C03634=1069.661,411.759,-112.459,175.801,35.006,156.496
C03635=1069.668,412.006,-112.501,175.806,35.015,156.498
C03636=1069.676,412.252,-112.545,175.812,35.025,156.501
C03637=1069.684,412.498,-112.589,175.818,35.034,156.503
C03638=1069.691,412.744,-112.631,175.824,35.044,156.505
C03639=1069.699,412.990,-112.675,175.831,35.054,156.508
C03640=1069.707,413.237,-112.719,175.837,35.064,156.510
C03641=1069.715,413.514,-112.768,175.844,35.074,156.512
C03642=1069.725,413.793,-112.817,175.850,35.085,156.515
C03643=1069.734,414.072,-112.867,175.857,35.096,156.518
C03644=1069.742,414.350,-112.916,175.864,35.108,156.520
C03645=1069.751,414.596,-112.959,175.870,35.117,156.523
C03646=1069.759,414.842,-113.003,175.877,35.127,156.525
C03647=1069.766,415.088,-113.047,175.883,35.137,156.527
C03648=1069.774,415.334,-113.091,175.888,35.147,156.530
C03649=1069.782,415.580,-113.135,175.894,35.157,156.532
C03650=1069.789,415.826,-113.178,175.901,35.167,156.535
C03651=1069.797,416.072,-113.222,175.907,35.177,156.537
C03652=1069.804,416.319,-113.267,175.913,35.187,156.539
C03653=1069.813,416.564,-113.311,175.919,35.197,156.542
C03654=1069.820,416.811,-113.354,175.926,35.208,156.544
C03655=1069.828,417.056,-113.399,175.932,35.218,156.547
C03656=1069.836,417.302,-113.443,175.938,35.228,156.549
C03657=1069.844,417.549,-113.487,175.944,35.238,156.552
C03658=1069.852,417.794,-113.531,175.951,35.248,156.554
C03659=1069.860,418.040,-113.575,175.957,35.259,156.557
C03660=1069.868,418.286,-113.620,175.963,35.269,156.559
C03661=1069.875,418.532,-113.664,175.970,35.279,156.562
C03662=1069.883,418.778,-113.708,175.976,35.290,156.564
C03663=1069.892,419.024,-113.753,175.983,35.300,156.567
C03664=1069.900,419.270,-113.797,175.989,35.310,156.569
C03665=1069.908,419.515,-113.841,175.995,35.321,156.572
C03666=1069.916,419.761,-113.886,176.003,35.331,156.574
C03667=1069.924,420.007,-113.930,176.009,35.342,156.577
C03668=1069.932,420.254,-113.975,176.016,35.353,156.579
C03669=1069.940,420.499,-114.020,176.022,35.363,156.582
C03670=1069.948,420.745,-114.064,176.029,35.373,156.584
C03671=1069.956,420.991,-114.108,176.035,35.384,156.587
C03672=1069.964,421.238,-114.154,176.042,35.395,156.590
C03673=1069.972,421.483,-114.199,176.048,35.406,156.592
C03674=1069.980,421.729,-114.243,176.055,35.417,156.595
C03675=1069.988,421.975,-114.288,176.062,35.427,156.598
C03676=1069.996,422.220,-114.333,176.069,35.438,156.600
C03677=1070.004,422.466,-114.378,176.075,35.449,156.603
C03678=1070.012,422.712,-114.423,176.082,35.460,156.606
C03679=1070.020,422.957,-114.468,176.088,35.471,156.608
C03680=1070.028,423.203,-114.513,176.095,35.482,156.611
C03681=1070.037,423.449,-114.558,176.102,35.493,156.614
C03682=1070.044,423.695,-114.604,176.109,35.504,156.616
C03683=1070.052,423.940,-114.648,176.115,35.515,156.619
C03684=1070.061,424.187,-114.694,176.122,35.526,156.622
C03685=1070.069,424.432,-114.739,176.130,35.537,156.625
C03686=1070.076,424.678,-114.784,176.136,35.548,156.627
C03687=1070.085,424.924,-114.829,176.143,35.559,156.630
C03688=1070.093,425.169,-114.875,176.150,35.571,156.633
C03689=1070.102,425.415,-114.920,176.157,35.582,156.636
C03690=1070.110,425.660,-114.966,176.164,35.593,156.638
C03691=1070.118,425.907,-115.011,176.171,35.604,156.641
C03692=1070.126,426.152,-115.056,176.177,35.615,156.644
C03693=1070.135,426.398,-115.102,176.185,35.627,156.647
C03694=1070.143,426.643,-115.148,176.192,35.638,156.650
C03695=1070.152,426.889,-115.193,176.199,35.650,156.652
C03696=1070.159,427.135,-115.239,176.206,35.661,156.655
C03697=1070.170,427.431,-115.294,176.214,35.675,156.659
C03698=1070.179,427.729,-115.350,176.223,35.689,156.662
C03699=1070.190,428.026,-115.405,176.232,35.703,156.666
C03700=1070.199,428.324,-115.461,176.240,35.717,156.669
C03701=1070.208,428.570,-115.507,176.248,35.729,156.672
C03702=1070.217,428.815,-115.553,176.255,35.741,156.675
C03703=1070.224,429.061,-115.599,176.263,35.753,156.678
C03704=1070.233,429.306,-115.645,176.270,35.764,156.681
C03705=1070.241,429.552,-115.691,176.277,35.776,156.684
C03706=1070.250,429.797,-115.737,176.285,35.788,156.687
C03707=1070.258,430.043,-115.783,176.291,35.800,156.690
C03708=1070.267,430.288,-115.830,176.299,35.812,156.693
C03709=1070.275,430.534,-115.877,176.306,35.824,156.696
C03710=1070.283,430.779,-115.922,176.314,35.836,156.699
C03711=1070.292,431.025,-115.968,176.321,35.848,156.702
C03712=1070.301,431.270,-116.015,176.329,35.860,156.705
C03713=1070.309,431.516,-116.061,176.336,35.872,156.708
C03714=1070.318,431.762,-116.108,176.344,35.884,156.711
C03715=1070.326,432.007,-116.155,176.352,35.896,156.714
C03716=1070.334,432.252,-116.201,176.359,35.909,156.717
C03717=1070.343,432.498,-116.248,176.367,35.922,156.721
C03718=1070.351,432.743,-116.294,176.374,35.934,156.724
C03719=1070.360,432.989,-116.341,176.382,35.946,156.727
C03720=1070.368,433.234,-116.388,176.390,35.959,156.730
C03721=1070.377,433.479,-116.435,176.397,35.971,156.733
C03722=1070.386,433.725,-116.482,176.406,35.984,156.736
C03723=1070.393,433.970,-116.529,176.414,35.996,156.739
C03724=1070.402,434.216,-116.576,176.421,36.009,156.743
C03725=1070.411,434.461,-116.623,176.429,36.021,156.746
C03726=1070.419,434.706,-116.670,176.437,36.034,156.749
C03727=1070.428,434.952,-116.717,176.444,36.047,156.752
C03728=1070.437,435.197,-116.764,176.452,36.059,156.756
C03729=1070.445,435.442,-116.811,176.461,36.072,156.759
C03730=1070.454,435.687,-116.859,176.468,36.085,156.762
C03731=1070.463,435.933,-116.905,176.476,36.098,156.765
C03732=1070.471,436.178,-116.953,176.484,36.111,156.769
C03733=1070.480,436.423,-117.001,176.493,36.124,156.772
C03734=1070.489,436.669,-117.048,176.501,36.137,156.775
C03735=1070.498,436.914,-117.095,176.508,36.150,156.779
C03736=1070.506,437.159,-117.143,176.516,36.163,156.782
C03737=1070.515,437.404,-117.190,176.525,36.176,156.785
C03738=1070.525,437.649,-117.238,176.533,36.189,156.789
C03739=1070.533,437.894,-117.286,176.541,36.202,156.792
C03740=1070.541,438.140,-117.333,176.550,36.215,156.796
C03741=1070.551,438.386,-117.381,176.558,36.229,156.799
C03742=1070.560,438.630,-117.428,176.566,36.242,156.802
C03743=1070.568,438.875,-117.477,176.574,36.255,156.806
C03744=1070.578,439.121,-117.525,176.582,36.269,156.809
C03745=1070.586,439.365,-117.572,176.591,36.282,156.813
C03746=1070.595,439.611,-117.620,176.599,36.295,156.816
C03747=1070.604,439.856,-117.668,176.608,36.309,156.820
C03748=1070.612,440.101,-117.717,176.616,36.323,156.823
C03749=1070.622,440.346,-117.764,176.625,36.336,156.827
C03750=1070.631,440.591,-117.812,176.633,36.350,156.830
C03751=1070.640,440.837,-117.861,176.642,36.364,156.834
C03752=1070.649,441.082,-117.908,176.650,36.377,156.838
C03753=1070.657,441.314,-117.955,176.659,36.391,156.841
C03754=1070.665,441.548,-118.001,176.667,36.404,156.845
C03755=1070.674,441.781,-118.047,176.675,36.417,156.848
C03756=1070.683,442.015,-118.093,176.683,36.430,156.851
C03757=1070.692,442.248,-118.140,176.693,36.444,156.855
C03758=1070.700,442.481,-118.186,176.701,36.457,156.858
C03759=1070.708,442.715,-118.232,176.709,36.471,156.862
C03760=1070.717,442.948,-118.279,176.718,36.484,156.865
C03761=1070.727,443.193,-118.327,176.726,36.498,156.869
C03762=1070.736,443.438,-118.376,176.735,36.513,156.873
C03763=1070.745,443.682,-118.425,176.744,36.527,156.877
C03764=1070.754,443.927,-118.474,176.754,36.541,156.881
C03765=1070.764,444.172,-118.522,176.762,36.556,156.884
C03766=1070.773,444.418,-118.571,176.771,36.570,156.888
C03767=1070.781,444.662,-118.620,176.781,36.584,156.892
C03768=1070.790,444.908,-118.669,176.790,36.599,156.896
C03769=1070.800,445.152,-118.719,176.799,36.614,156.900
C03770=1070.809,445.397,-118.768,176.808,36.628,156.904
C03771=1070.819,445.642,-118.817,176.817,36.643,156.907
C03772=1070.828,445.887,-118.867,176.826,36.658,156.911
C03773=1070.837,446.132,-118.915,176.836,36.672,156.915
C03774=1070.846,446.376,-118.965,176.845,36.687,156.919
C03775=1070.855,446.621,-119.014,176.855,36.702,156.923
C03776=1070.864,446.866,-119.064,176.864,36.717,156.927
C03777=1070.874,447.111,-119.113,176.874,36.732,156.931
C03778=1070.884,447.355,-119.163,176.883,36.747,156.935
C03779=1070.893,447.601,-119.212,176.893,36.762,156.939
C03780=1070.903,447.846,-119.262,176.902,36.777,156.943
C03781=1070.913,448.089,-119.312,176.911,36.793,156.947
C03782=1070.922,448.332,-119.360,176.920,36.807,156.951
C03783=1070.932,448.577,-119.410,176.929,36.822,156.955
C03784=1070.944,448.821,-119.458,176.937,36.836,156.959
C03785=1070.957,449.066,-119.505,176.945,36.850,156.963
C03786=1070.972,449.311,-119.551,176.953,36.863,156.966
C03787=1070.987,449.556,-119.598,176.960,36.876,156.970
C03788=1071.004,449.802,-119.643,176.968,36.888,156.973
C03789=1070.654,449.802,-119.894,176.954,37.029,157.010
C03790=1070.638,449.556,-119.849,176.947,37.016,157.007
C03791=1070.622,449.311,-119.803,176.939,37.004,157.004
C03792=1070.608,449.066,-119.756,176.931,36.990,157.000
C03793=1070.595,448.821,-119.709,176.923,36.977,156.996
C03794=1070.582,448.576,-119.661,176.914,36.963,156.993
C03795=1070.571,448.332,-119.612,176.905,36.948,156.989
C03796=1070.562,448.088,-119.563,176.896,36.933,156.985
C03797=1070.553,447.845,-119.513,176.886,36.918,156.981
C03798=1070.543,447.601,-119.463,176.877,36.903,156.977
C03799=1070.533,447.356,-119.413,176.867,36.888,156.973
C03800=1070.523,447.111,-119.364,176.858,36.873,156.969
C03801=1070.514,446.866,-119.315,176.848,36.858,156.965
C03802=1070.505,446.621,-119.265,176.838,36.843,156.961
C03803=1070.496,446.376,-119.215,176.829,36.828,156.957
C03804=1070.486,446.131,-119.166,176.819,36.814,156.953
C03805=1070.477,445.887,-119.116,176.810,36.799,156.949
C03806=1070.468,445.641,-119.067,176.800,36.784,156.945
C03807=1070.458,445.397,-119.018,176.792,36.770,156.941
C03808=1070.449,445.153,-118.969,176.782,36.755,156.937
C03809=1070.440,444.908,-118.920,176.773,36.741,156.933
C03810=1070.431,444.663,-118.870,176.764,36.726,156.929
C03811=1070.422,444.417,-118.821,176.754,36.711,156.925
C03812=1070.412,444.173,-118.772,176.745,36.697,156.922
C03813=1070.403,443.928,-118.723,176.736,36.683,156.918
C03814=1070.394,443.683,-118.674,176.727,36.668,156.914
C03815=1070.384,443.438,-118.626,176.718,36.654,156.910
C03816=1070.375,443.193,-118.577,176.708,36.640,156.906
C03817=1070.366,442.949,-118.528,176.700,36.626,156.903
C03818=1070.358,442.724,-118.484,176.692,36.612,156.899
C03819=1070.349,442.500,-118.439,176.684,36.600,156.896
C03820=1070.341,442.276,-118.394,176.675,36.587,156.892
C03821=1070.333,442.052,-118.351,176.667,36.574,156.889
C03822=1070.324,441.828,-118.306,176.659,36.562,156.886
C03823=1070.316,441.604,-118.261,176.651,36.549,156.882
C03824=1070.308,441.380,-118.218,176.643,36.536,156.879
C03825=1070.300,441.156,-118.173,176.635,36.524,156.876
C03826=1070.291,440.912,-118.124,176.627,36.510,156.872
C03827=1070.282,440.666,-118.076,176.618,36.496,156.869
C03828=1070.273,440.421,-118.027,176.609,36.482,156.865
C03829=1070.264,440.176,-117.980,176.600,36.468,156.861
C03830=1070.254,439.931,-117.931,176.592,36.455,156.858
C03831=1070.246,439.686,-117.883,176.583,36.442,156.854
C03832=1070.237,439.441,-117.836,176.575,36.428,156.851
C03833=1070.228,439.195,-117.787,176.566,36.415,156.847
C03834=1070.219,438.951,-117.739,176.558,36.401,156.844
C03835=1070.210,438.705,-117.692,176.549,36.388,156.840
C03836=1070.202,438.460,-117.643,176.541,36.374,156.837
C03837=1070.193,438.215,-117.596,176.533,36.361,156.833
C03838=1070.183,437.969,-117.548,176.524,36.348,156.830
C03839=1070.174,437.724,-117.501,176.516,36.335,156.827
C03840=1070.166,437.480,-117.453,176.507,36.322,156.823
C03841=1070.157,437.234,-117.405,176.499,36.309,156.820
C03842=1070.148,436.989,-117.357,176.491,36.296,156.817
C03843=1070.139,436.744,-117.310,176.483,36.283,156.813
C03844=1070.130,436.498,-117.263,176.475,36.270,156.810
C03845=1070.121,436.253,-117.215,176.467,36.257,156.807
C03846=1070.112,436.008,-117.168,176.459,36.244,156.803
C03847=1070.104,435.762,-117.121,176.450,36.231,156.800
C03848=1070.096,435.517,-117.073,176.442,36.218,156.797
C03849=1070.087,435.272,-117.026,176.434,36.205,156.793
C03850=1070.078,435.027,-116.979,176.427,36.193,156.790
C03851=1070.069,434.781,-116.931,176.419,36.180,156.787
C03852=1070.060,434.536,-116.885,176.410,36.167,156.784
C03853=1070.051,434.291,-116.837,176.402,36.155,156.780
C03854=1070.043,434.045,-116.790,176.395,36.142,156.777
C03855=1070.034,433.800,-116.744,176.387,36.130,156.774
C03856=1070.026,433.554,-116.697,176.379,36.117,156.771
C03857=1070.017,433.309,-116.649,176.371,36.105,156.768
C03858=1070.008,433.064,-116.603,176.364,36.092,156.764
C03859=1070.001,432.818,-116.555,176.356,36.080,156.761
C03860=1069.992,432.572,-116.509,176.348,36.068,156.758
C03861=1069.984,432.328,-116.462,176.341,36.055,156.755
C03862=1069.976,432.082,-116.416,176.333,36.043,156.752
C03863=1069.967,431.837,-116.369,176.325,36.031,156.749
C03864=1069.958,431.591,-116.322,176.318,36.018,156.746
C03865=1069.950,431.346,-116.275,176.310,36.006,156.743
C03866=1069.941,431.100,-116.229,176.303,35.994,156.740
C03867=1069.932,430.855,-116.183,176.295,35.982,156.737
C03868=1069.924,430.609,-116.137,176.287,35.970,156.734
C03869=1069.916,430.364,-116.090,176.280,35.958,156.730
C03870=1069.907,430.118,-116.043,176.272,35.946,156.727
C03871=1069.898,429.873,-115.998,176.265,35.934,156.724
C03872=1069.890,429.627,-115.951,176.257,35.923,156.721
C03873=1069.882,429.382,-115.905,176.250,35.910,156.718
C03874=1069.874,429.136,-115.859,176.242,35.899,156.716
C03875=1069.865,428.891,-115.812,176.235,35.887,156.713
C03876=1069.857,428.645,-115.767,176.228,35.875,156.710
C03877=1069.849,428.399,-115.721,176.221,35.864,156.707
C03878=1069.838,428.100,-115.665,176.212,35.849,156.703
C03879=1069.829,427.801,-115.609,176.203,35.835,156.700
C03880=1069.818,427.503,-115.553,176.194,35.821,156.696
C03881=1069.808,427.203,-115.497,176.185,35.807,156.693
C03882=1069.800,426.957,-115.451,176.178,35.796,156.690
C03883=1069.791,426.712,-115.406,176.171,35.784,156.687
C03884=1069.783,426.466,-115.360,176.164,35.773,156.684
C03885=1069.775,426.220,-115.315,176.156,35.761,156.681
C03886=1069.766,425.974,-115.269,176.150,35.750,156.678
C03887=1069.758,425.729,-115.224,176.142,35.739,156.676
C03888=1069.750,425.483,-115.178,176.135,35.728,156.673
C03889=1069.741,425.238,-115.133,176.129,35.716,156.670
C03890=1069.733,424.992,-115.087,176.121,35.705,156.667
C03891=1069.725,424.747,-115.042,176.114,35.694,156.665
C03892=1069.717,424.501,-114.996,176.108,35.683,156.662
C03893=1069.709,424.255,-114.951,176.101,35.672,156.659
C03894=1069.701,424.009,-114.906,176.093,35.661,156.656
C03895=1069.692,423.764,-114.860,176.087,35.650,156.654
C03896=1069.685,423.517,-114.815,176.080,35.639,156.651
C03897=1069.676,423.272,-114.770,176.073,35.628,156.648
C03898=1069.667,423.027,-114.725,176.066,35.617,156.645
C03899=1069.660,422.780,-114.680,176.060,35.606,156.643
C03900=1069.652,422.535,-114.635,176.053,35.595,156.640
C03901=1069.644,422.289,-114.590,176.045,35.584,156.637
C03902=1069.635,422.043,-114.545,176.039,35.573,156.635
C03903=1069.628,421.797,-114.500,176.032,35.563,156.632
C03904=1069.620,421.552,-114.455,176.026,35.552,156.629
C03905=1069.611,421.306,-114.410,176.019,35.541,156.627
C03906=1069.604,421.060,-114.365,176.012,35.530,156.624
C03907=1069.595,420.814,-114.321,176.005,35.520,156.622
C03908=1069.587,420.568,-114.276,175.999,35.509,156.619
C03909=1069.579,420.322,-114.232,175.993,35.499,156.616
C03910=1069.571,420.076,-114.187,175.986,35.488,156.614
C03911=1069.563,419.831,-114.142,175.980,35.477,156.611
C03912=1069.555,419.585,-114.097,175.973,35.467,156.609
C03913=1069.547,419.339,-114.053,175.966,35.457,156.606
C03914=1069.539,419.093,-114.009,175.959,35.446,156.604
C03915=1069.530,418.846,-113.965,175.953,35.436,156.601
C03916=1069.522,418.601,-113.920,175.947,35.426,156.599
C03917=1069.515,418.355,-113.875,175.940,35.416,156.596
C03918=1069.507,418.109,-113.831,175.934,35.405,156.594
C03919=1069.499,417.863,-113.787,175.928,35.395,156.591
C03920=1069.491,417.617,-113.742,175.921,35.384,156.589
C03921=1069.483,417.371,-113.699,175.915,35.374,156.586
C03922=1069.475,417.125,-113.654,175.909,35.364,156.584
C03923=1069.467,416.879,-113.610,175.902,35.354,156.581
C03924=1069.459,416.633,-113.566,175.896,35.344,156.579
C03925=1069.451,416.387,-113.522,175.890,35.334,156.576
C03926=1069.444,416.141,-113.477,175.883,35.323,156.574
C03927=1069.437,415.896,-113.434,175.876,35.313,156.571
C03928=1069.429,415.650,-113.390,175.870,35.304,156.569
C03929=1069.421,415.404,-113.346,175.864,35.293,156.567
C03930=1069.413,415.158,-113.302,175.859,35.284,156.564
C03931=1069.405,414.911,-113.258,175.851,35.274,156.562
C03932=1069.397,414.665,-113.214,175.846,35.264,156.560
C03933=1069.389,414.419,-113.170,175.840,35.254,156.557
C03934=1069.380,414.139,-113.121,175.832,35.243,156.554
C03935=1069.371,413.859,-113.071,175.825,35.232,156.552
C03936=1069.362,413.579,-113.021,175.818,35.220,156.549
C03937=1069.353,413.298,-112.972,175.811,35.210,156.546
C03938=1069.346,413.053,-112.928,175.805,35.200,156.544
C03939=1069.337,412.807,-112.885,175.799,35.190,156.542
C03940=1069.329,412.561,-112.842,175.793,35.180,156.540
C03941=1069.322,412.314,-112.798,175.788,35.171,156.537
C03942=1069.314,412.069,-112.755,175.782,35.162,156.535
C03943=1069.306,411.823,-112.712,175.776,35.152,156.533
C03944=1069.298,411.576,-112.668,175.770,35.142,156.530
C03945=1069.290,411.330,-112.625,175.764,35.133,156.528
C03946=1069.284,411.084,-112.582,175.757,35.123,156.526
C03947=1069.275,410.838,-112.539,175.751,35.113,156.524
C03948=1069.267,410.591,-112.495,175.745,35.104,156.521
C03949=1069.260,410.346,-112.452,175.740,35.095,156.519
C03950=1069.252,410.099,-112.409,175.734,35.085,156.517
C03951=1069.245,409.853,-112.367,175.728,35.076,156.515
C03952=1069.237,409.607,-112.323,175.722,35.067,156.513
C03953=1069.230,409.361,-112.280,175.716,35.057,156.510
C03954=1069.222,409.115,-112.237,175.710,35.048,156.508
C03955=1069.214,408.868,-112.194,175.704,35.039,156.506
C03956=1069.207,408.622,-112.151,175.699,35.030,156.504
C03957=1069.199,408.376,-112.108,175.693,35.020,156.502
C03958=1069.191,408.130,-112.065,175.687,35.011,156.499
C03959=1069.184,407.884,-112.023,175.682,35.002,156.497
C03960=1069.176,407.637,-111.980,175.676,34.993,156.495
C03961=1069.169,407.392,-111.937,175.671,34.984,156.493
C03962=1069.161,407.145,-111.895,175.665,34.975,156.491
C03963=1069.154,406.899,-111.851,175.659,34.966,156.489
C03964=1069.146,406.652,-111.808,175.653,34.956,156.486
C03965=1069.139,406.406,-111.766,175.648,34.948,156.484
C03966=1069.132,406.161,-111.723,175.642,34.938,156.482
C03967=1069.123,405.914,-111.681,175.636,34.930,156.480
C03968=1069.117,405.668,-111.638,175.631,34.921,156.478
C03969=1069.109,405.422,-111.596,175.626,34.912,156.476
C03970=1069.102,405.175,-111.554,175.620,34.903,156.474
C03971=1069.094,404.929,-111.512,175.614,34.894,156.472
C03972=1069.086,404.683,-111.470,175.608,34.885,156.470
C03973=1069.079,404.436,-111.427,175.603,34.876,156.468
C03974=1069.071,404.190,-111.385,175.598,34.868,156.466
C03975=1069.064,403.943,-111.342,175.592,34.859,156.464
C03976=1069.056,403.697,-111.300,175.587,34.850,156.462
C03977=1069.049,403.451,-111.258,175.581,34.841,156.460
C03978=1069.042,403.204,-111.215,175.575,34.833,156.458
C03979=1069.034,402.959,-111.173,175.570,34.824,156.455
C03980=1069.027,402.713,-111.132,175.565,34.815,156.453
C03981=1069.018,402.466,-111.089,175.559,34.807,156.451
C03982=1069.012,402.219,-111.047,175.553,34.798,156.449
C03983=1069.004,401.973,-111.005,175.549,34.790,156.447
C03984=1068.997,401.727,-110.964,175.543,34.781,156.445
C03985=1068.989,401.481,-110.922,175.537,34.773,156.444
C03986=1068.981,401.234,-110.880,175.532,34.764,156.442
C03987=1068.974,400.987,-110.837,175.527,34.756,156.440
C03988=1068.967,400.741,-110.796,175.521,34.747,156.438
C03989=1068.959,400.495,-110.754,175.516,34.739,156.436
C03990=1068.951,400.219,-110.707,175.510,34.729,156.434
C03991=1068.943,399.942,-110.661,175.504,34.719,156.431
C03992=1068.935,399.666,-110.614,175.498,34.710,156.429
C03993=1068.926,399.390,-110.567,175.492,34.701,156.427
C03994=1068.919,399.143,-110.526,175.487,34.693,156.425
C03995=1068.912,398.897,-110.484,175.482,34.684,156.423
C03996=1068.904,398.651,-110.442,175.476,34.676,156.421
C03997=1068.897,398.404,-110.401,175.472,34.668,156.419
C03998=1068.889,398.158,-110.359,175.466,34.660,156.417
C03999=1068.882,397.912,-110.318,175.460,34.651,156.416
C04000=1068.875,397.665,-110.277,175.456,34.643,156.414
C04001=1068.867,397.418,-110.235,175.450,34.635,156.412
C04002=1068.860,397.172,-110.194,175.445,34.627,156.410
C04003=1068.853,396.926,-110.152,175.440,34.618,156.408
C04004=1068.846,396.680,-110.111,175.434,34.611,156.406
C04005=1068.839,396.433,-110.070,175.430,34.602,156.404
C04006=1068.831,396.187,-110.029,175.424,34.594,156.402
C04007=1068.824,395.940,-109.988,175.420,34.586,156.401
C04008=1068.817,395.694,-109.947,175.414,34.578,156.399
C04009=1068.809,395.447,-109.905,175.409,34.570,156.397
C04010=1068.801,395.201,-109.865,175.404,34.562,156.395
C04011=1068.795,394.955,-109.824,175.399,34.554,156.393
C04012=1068.787,394.708,-109.783,175.394,34.546,156.391
C04013=1068.780,394.462,-109.741,175.389,34.538,156.390
C04014=1068.773,394.215,-109.700,175.384,34.531,156.388
C04015=1068.766,393.969,-109.659,175.378,34.522,156.386
C04016=1068.759,393.722,-109.619,175.374,34.515,156.384
C04017=1068.751,393.476,-109.578,175.368,34.507,156.383
C04018=1068.744,393.229,-109.537,175.364,34.499,156.381
C04019=1068.737,392.983,-109.496,175.358,34.491,156.379
C04020=1068.730,392.736,-109.455,175.353,34.484,156.377
C04021=1068.722,392.490,-109.415,175.348,34.476,156.376
C04022=1068.716,392.244,-109.374,175.343,34.468,156.374
C04023=1068.709,391.997,-109.333,175.338,34.460,156.372
C04024=1068.701,391.750,-109.293,175.334,34.453,156.370
C04025=1068.694,391.504,-109.252,175.328,34.445,156.369
C04026=1068.687,391.257,-109.211,175.324,34.437,156.367
C04027=1068.679,391.011,-109.171,175.318,34.429,156.365
C04028=1068.672,390.764,-109.131,175.314,34.422,156.363
C04029=1068.665,390.518,-109.089,175.309,34.414,156.362
C04030=1068.658,390.272,-109.050,175.304,34.407,156.360
C04031=1068.651,390.025,-109.009,175.299,34.399,156.358
C04032=1068.643,389.778,-108.969,175.294,34.392,156.356
C04033=1068.637,389.532,-108.929,175.289,34.384,156.355
C04034=1068.629,389.285,-108.888,175.284,34.376,156.353
C04035=1068.622,389.039,-108.848,175.279,34.369,156.351
C04036=1068.615,388.792,-108.808,175.274,34.361,156.350
C04037=1068.607,388.546,-108.768,175.270,34.354,156.348
C04038=1068.600,388.299,-108.727,175.264,34.346,156.346
C04039=1068.592,388.052,-108.687,175.260,34.339,156.345
C04040=1068.586,387.806,-108.647,175.255,34.332,156.343
C04041=1068.579,387.559,-108.608,175.250,34.325,156.341
C04042=1068.571,387.313,-108.568,175.246,34.317,156.340
C04043=1068.564,387.067,-108.527,175.240,34.310,156.338
C04044=1068.557,386.820,-108.487,175.236,34.302,156.337
C04045=1068.550,386.573,-108.447,175.231,34.295,156.335
C04046=1068.542,386.313,-108.405,175.226,34.287,156.333
C04047=1068.535,386.052,-108.363,175.221,34.279,156.331
C04048=1068.528,385.792,-108.320,175.216,34.272,156.330
C04049=1068.521,385.532,-108.278,175.211,34.264,156.328
C04050=1068.513,385.285,-108.239,175.206,34.257,156.326
C04051=1068.506,385.038,-108.199,175.201,34.250,156.325
C04052=1068.499,384.792,-108.159,175.197,34.243,156.323
C04053=1068.492,384.546,-108.119,175.192,34.235,156.322
C04054=1068.485,384.301,-108.079,175.188,34.228,156.320
C04055=1068.478,384.056,-108.041,175.182,34.221,156.318
C04056=1068.471,383.811,-108.001,175.178,34.214,156.317
C04057=1068.464,383.567,-107.962,175.174,34.207,156.315
C04058=1068.458,383.322,-107.922,175.168,34.200,156.314
C04059=1068.450,383.078,-107.883,175.164,34.193,156.312
C04060=1068.444,382.833,-107.844,175.160,34.186,156.311
C04061=1068.436,382.588,-107.804,175.155,34.179,156.309
C04062=1068.430,382.342,-107.764,175.151,34.171,156.307
C04063=1068.423,382.095,-107.725,175.146,34.165,156.306
C04064=1068.416,381.849,-107.686,175.141,34.157,156.304
C04065=1068.409,381.601,-107.646,175.137,34.151,156.303
C04066=1068.402,381.355,-107.607,175.132,34.143,156.301
C04067=1068.396,381.108,-107.568,175.127,34.137,156.300
C04068=1068.388,380.862,-107.528,175.123,34.129,156.298
C04069=1068.381,380.614,-107.489,175.118,34.123,156.297
C04070=1068.374,380.368,-107.449,175.114,34.116,156.295
C04071=1068.367,380.121,-107.411,175.109,34.109,156.294
C04072=1068.360,379.874,-107.372,175.104,34.102,156.292
C04073=1068.353,379.628,-107.332,175.100,34.095,156.291
C04074=1068.346,379.381,-107.293,175.096,34.088,156.289
C04075=1068.339,379.134,-107.254,175.090,34.081,156.288
C04076=1068.332,378.888,-107.215,175.086,34.075,156.286
C04077=1068.325,378.641,-107.176,175.082,34.068,156.285
C04078=1068.318,378.394,-107.137,175.077,34.061,156.283
C04079=1068.311,378.147,-107.098,175.073,34.054,156.282
C04080=1068.305,377.900,-107.059,175.068,34.048,156.280
C04081=1068.297,377.654,-107.020,175.064,34.041,156.279
C04082=1068.290,377.407,-106.980,175.059,34.034,156.277
C04083=1068.283,377.160,-106.942,175.055,34.027,156.276
C04084=1068.276,376.913,-106.903,175.051,34.021,156.274
C04085=1068.270,376.666,-106.864,175.046,34.014,156.273
C04086=1068.263,376.419,-106.825,175.041,34.007,156.271
C04087=1068.256,376.172,-106.786,175.037,34.001,156.270
C04088=1068.249,375.926,-106.747,175.032,33.994,156.268
C04089=1068.242,375.679,-106.709,175.028,33.987,156.267
C04090=1068.236,375.432,-106.670,175.024,33.981,156.266
C04091=1068.229,375.185,-106.631,175.020,33.974,156.264
C04092=1068.222,374.938,-106.592,175.015,33.967,156.263
C04093=1068.215,374.691,-106.554,175.011,33.961,156.261
C04094=1068.209,374.444,-106.515,175.007,33.954,156.260
C04095=1068.202,374.197,-106.476,175.001,33.947,156.258
C04096=1068.195,373.951,-106.438,174.997,33.941,156.257
C04097=1068.188,373.705,-106.400,174.993,33.934,156.256
C04098=1068.182,373.464,-106.362,174.989,33.928,156.254
C04099=1068.175,373.223,-106.324,174.984,33.922,156.253
C04100=1068.169,372.983,-106.286,174.980,33.915,156.251
C04101=1068.162,372.742,-106.250,174.976,33.909,156.250
C04102=1068.155,372.501,-106.212,174.972,33.903,156.249
C04103=1068.148,372.261,-106.175,174.967,33.896,156.247
C04104=1068.141,372.020,-106.138,174.963,33.890,156.246
C04105=1068.135,371.780,-106.100,174.959,33.884,156.245
C04106=1068.128,371.533,-106.062,174.955,33.878,156.243
C04107=1068.121,371.286,-106.024,174.950,33.871,156.242
C04108=1068.114,371.039,-105.986,174.946,33.865,156.241
C04109=1068.107,370.792,-105.947,174.942,33.859,156.239
C04110=1068.101,370.545,-105.909,174.938,33.853,156.238
C04111=1068.093,370.298,-105.871,174.933,33.846,156.237
C04112=1068.087,370.051,-105.833,174.929,33.840,156.235
C04113=1068.080,369.805,-105.795,174.925,33.833,156.234
C04114=1068.073,369.558,-105.757,174.921,33.827,156.232
C04115=1068.067,369.310,-105.719,174.917,33.821,156.231
C04116=1068.059,369.064,-105.680,174.912,33.814,156.230
C04117=1068.053,368.816,-105.642,174.908,33.808,156.228
C04118=1068.046,368.570,-105.605,174.904,33.802,156.227
C04119=1068.040,368.322,-105.567,174.900,33.796,156.226
C04120=1068.033,368.076,-105.528,174.895,33.790,156.224
C04121=1068.026,367.828,-105.491,174.891,33.784,156.223
C04122=1068.020,367.582,-105.453,174.887,33.777,156.222
C04123=1068.012,367.335,-105.415,174.883,33.771,156.220
C04124=1068.006,367.087,-105.377,174.879,33.765,156.219
C04125=1067.999,366.841,-105.340,174.874,33.758,156.218
C04126=1067.992,366.594,-105.301,174.870,33.753,156.217
C04127=1067.985,366.347,-105.264,174.866,33.746,156.215
C04128=1067.979,366.100,-105.226,174.862,33.740,156.214
C04129=1067.972,365.853,-105.188,174.857,33.734,156.213
C04130=1067.966,365.605,-105.150,174.853,33.728,156.211
C04131=1067.959,365.359,-105.113,174.849,33.722,156.210
C04132=1067.952,365.112,-105.075,174.845,33.715,156.209
C04133=1067.946,364.865,-105.038,174.841,33.710,156.207
C04134=1067.939,364.618,-105.000,174.838,33.703,156.206
C04135=1067.932,364.370,-104.963,174.833,33.698,156.205
C04136=1067.926,364.123,-104.925,174.829,33.691,156.204
C04137=1067.919,363.876,-104.888,174.825,33.686,156.202
C04138=1067.912,363.629,-104.850,174.821,33.679,156.201
C04139=1067.906,363.382,-104.812,174.817,33.674,156.200
C04140=1067.899,363.135,-104.775,174.812,33.667,156.198
C04141=1067.892,362.888,-104.738,174.808,33.662,156.197
C04142=1067.885,362.641,-104.701,174.804,33.656,156.196
C04143=1067.879,362.394,-104.663,174.800,33.649,156.195
C04144=1067.872,362.146,-104.626,174.796,33.644,156.193
C04145=1067.865,361.899,-104.589,174.793,33.638,156.192
C04146=1067.858,361.653,-104.552,174.788,33.632,156.191
C04147=1067.852,361.405,-104.514,174.784,33.626,156.190
C04148=1067.846,361.158,-104.477,174.780,33.620,156.188
C04149=1067.839,360.910,-104.440,174.776,33.614,156.187
C04150=1067.832,360.664,-104.403,174.772,33.609,156.186
C04151=1067.825,360.417,-104.366,174.768,33.603,156.185
C04152=1067.819,360.170,-104.329,174.763,33.596,156.184
C04153=1067.812,359.922,-104.291,174.760,33.591,156.182
C04154=1067.805,359.692,-104.257,174.756,33.586,156.181
C04155=1067.800,359.463,-104.223,174.752,33.580,156.180
C04156=1067.794,359.233,-104.189,174.749,33.575,156.179
C04157=1067.788,359.003,-104.154,174.745,33.569,156.178
C04158=1067.782,358.773,-104.119,174.742,33.564,156.177
C04159=1067.776,358.543,-104.085,174.737,33.558,156.176
C04160=1067.769,358.313,-104.051,174.733,33.553,156.174
C04161=1067.763,358.084,-104.016,174.730,33.548,156.173
C04162=1067.757,357.837,-103.979,174.726,33.542,156.172
C04163=1067.750,357.589,-103.943,174.722,33.536,156.171
C04164=1067.743,357.342,-103.906,174.718,33.531,156.170
C04165=1067.736,357.095,-103.869,174.715,33.525,156.169
C04166=1067.730,356.848,-103.832,174.710,33.519,156.167
C04167=1067.723,356.600,-103.796,174.706,33.514,156.166
C04168=1067.717,356.353,-103.759,174.702,33.508,156.165
C04169=1067.710,356.106,-103.723,174.698,33.502,156.164
C04170=1067.703,355.858,-103.686,174.695,33.497,156.163
C04171=1067.697,355.611,-103.649,174.691,33.491,156.162
C04172=1067.690,355.364,-103.612,174.687,33.485,156.160
C04173=1067.684,355.117,-103.576,174.683,33.480,156.159
C04174=1067.677,354.870,-103.539,174.678,33.474,156.158
C04175=1067.671,354.623,-103.502,174.675,33.469,156.157
C04176=1067.664,354.375,-103.466,174.671,33.463,156.156
C04177=1067.657,354.128,-103.430,174.667,33.457,156.154
C04178=1067.650,353.881,-103.393,174.663,33.452,156.153
C04179=1067.644,353.634,-103.357,174.660,33.446,156.152
C04180=1067.638,353.387,-103.320,174.656,33.440,156.151
C04181=1067.631,353.139,-103.284,174.652,33.435,156.150
C04182=1067.624,352.892,-103.247,174.647,33.429,156.149
C04183=1067.618,352.644,-103.211,174.644,33.424,156.148
C04184=1067.612,352.397,-103.175,174.640,33.418,156.146
C04185=1067.605,352.150,-103.138,174.636,33.413,156.145
C04186=1067.599,351.903,-103.102,174.633,33.407,156.144
C04187=1067.592,351.656,-103.066,174.629,33.402,156.143
C04188=1067.586,351.408,-103.030,174.625,33.397,156.142
C04189=1067.579,351.161,-102.994,174.621,33.391,156.141
C04190=1067.572,350.913,-102.957,174.618,33.386,156.140
C04191=1067.565,350.667,-102.921,174.613,33.380,156.138
C04192=1067.559,350.419,-102.885,174.609,33.374,156.137
C04193=1067.553,350.172,-102.849,174.605,33.369,156.136
C04194=1067.546,349.924,-102.814,174.602,33.364,156.135
C04195=1067.539,349.677,-102.777,174.598,33.358,156.134
C04196=1067.533,349.430,-102.740,174.594,33.353,156.133
C04197=1067.526,349.182,-102.705,174.591,33.348,156.132
C04198=1067.520,348.935,-102.669,174.587,33.342,156.131
C04199=1067.514,348.688,-102.633,174.583,33.337,156.130
C04200=1067.507,348.440,-102.597,174.580,33.331,156.129
C04201=1067.501,348.193,-102.562,174.576,33.326,156.127
C04202=1067.494,347.946,-102.525,174.571,33.321,156.126
C04203=1067.488,347.698,-102.489,174.568,33.316,156.125
C04204=1067.481,347.451,-102.453,174.564,33.310,156.124
C04205=1067.475,347.203,-102.417,174.560,33.304,156.123
C04206=1067.467,346.957,-102.382,174.557,33.299,156.122
C04207=1067.461,346.709,-102.346,174.553,33.294,156.121
C04208=1067.455,346.461,-102.310,174.549,33.289,156.120
C04209=1067.448,346.214,-102.274,174.546,33.283,156.119
C04210=1067.442,345.986,-102.242,174.542,33.279,156.118
C04211=1067.436,345.758,-102.209,174.539,33.273,156.117
C04212=1067.431,345.531,-102.176,174.536,33.269,156.116
C04213=1067.425,345.303,-102.143,174.532,33.264,156.115
C04214=1067.419,345.074,-102.110,174.529,33.259,156.114
C04215=1067.413,344.846,-102.078,174.525,33.254,156.113
C04216=1067.407,344.619,-102.044,174.521,33.249,156.112
C04217=1067.401,344.390,-102.012,174.518,33.245,156.111
C04218=1067.395,344.143,-101.976,174.514,33.239,156.110
C04219=1067.388,343.895,-101.941,174.511,33.234,156.109
C04220=1067.382,343.648,-101.905,174.507,33.229,156.108
C04221=1067.375,343.400,-101.870,174.504,33.224,156.107
C04222=1067.368,343.154,-101.834,174.500,33.218,156.105
C04223=1067.363,342.907,-101.799,174.496,33.213,156.104
C04224=1067.356,342.659,-101.764,174.493,33.208,156.103
C04225=1067.349,342.412,-101.728,174.489,33.203,156.102
C04226=1067.343,342.164,-101.693,174.486,33.198,156.101
C04227=1067.336,341.917,-101.658,174.482,33.192,156.100
C04228=1067.330,341.670,-101.622,174.478,33.188,156.099
C04229=1067.324,341.422,-101.587,174.475,33.182,156.098
C04230=1067.317,341.175,-101.552,174.471,33.177,156.097
C04231=1067.310,340.927,-101.517,174.468,33.172,156.096
C04232=1067.304,340.679,-101.481,174.464,33.167,156.095
C04233=1067.298,340.431,-101.446,174.460,33.162,156.094
C04234=1067.291,340.184,-101.411,174.456,33.157,156.093
C04235=1067.285,339.937,-101.376,174.452,33.152,156.092
C04236=1067.279,339.690,-101.341,174.449,33.146,156.091
C04237=1067.272,339.442,-101.306,174.445,33.142,156.090
C04238=1067.265,339.194,-101.271,174.442,33.136,156.089
C04239=1067.259,338.947,-101.235,174.438,33.132,156.088
C04240=1067.253,338.699,-101.200,174.435,33.126,156.087
C04241=1067.246,338.453,-101.166,174.431,33.121,156.086
C04242=1067.241,338.204,-101.130,174.428,33.116,156.085
C04243=1067.234,337.957,-101.095,174.424,33.111,156.084
C04244=1067.227,337.710,-101.060,174.421,33.106,156.083
C04245=1067.221,337.462,-101.026,174.417,33.101,156.082
C04246=1067.215,337.215,-100.991,174.414,33.096,156.081
C04247=1067.208,336.967,-100.955,174.410,33.091,156.080
C04248=1067.202,336.719,-100.921,174.407,33.086,156.079
C04249=1067.195,336.472,-100.886,174.403,33.081,156.078
C04250=1067.189,336.225,-100.852,174.400,33.076,156.077
C04251=1067.183,335.977,-100.817,174.396,33.071,156.076
C04252=1067.176,335.729,-100.782,174.393,33.066,156.075
C04253=1067.169,335.482,-100.747,174.389,33.061,156.074
C04254=1067.164,335.235,-100.713,174.386,33.057,156.073
C04255=1067.157,334.987,-100.678,174.382,33.051,156.072
C04256=1067.150,334.739,-100.643,174.379,33.047,156.071
C04257=1067.144,334.492,-100.608,174.375,33.042,156.070
C04258=1067.138,334.245,-100.574,174.372,33.037,156.069
C04259=1067.131,333.997,-100.540,174.368,33.032,156.068
C04260=1067.124,333.749,-100.505,174.365,33.027,156.067
C04261=1067.119,333.502,-100.471,174.361,33.022,156.066
C04262=1067.112,333.254,-100.436,174.357,33.017,156.065
C04263=1067.105,333.007,-100.401,174.353,33.012,156.064
C04264=1067.099,332.759,-100.367,174.350,33.007,156.063
C04265=1067.093,332.511,-100.333,174.347,33.003,156.062
C04266=1067.088,332.281,-100.300,174.343,32.998,156.061
C04267=1067.081,332.051,-100.268,174.340,32.993,156.060
C04268=1067.076,331.820,-100.236,174.337,32.989,156.060
C04269=1067.070,331.590,-100.204,174.334,32.984,156.059
C04270=1067.064,331.360,-100.172,174.331,32.980,156.058
C04271=1067.058,331.129,-100.140,174.327,32.975,156.057
C04272=1067.052,330.899,-100.109,174.324,32.971,156.056
C04273=1067.046,330.668,-100.076,174.321,32.966,156.055
C04274=1067.040,330.421,-100.043,174.318,32.962,156.054
C04275=1067.033,330.173,-100.008,174.314,32.957,156.053
C04276=1067.027,329.925,-99.974,174.311,32.952,156.052
C04277=1067.020,329.679,-99.940,174.307,32.947,156.051
C04278=1067.013,329.431,-99.905,174.304,32.943,156.050
C04279=1067.007,329.183,-99.871,174.300,32.938,156.049
C04280=1067.000,328.936,-99.838,174.297,32.933,156.048
C04281=1066.994,328.687,-99.804,174.294,32.928,156.048
C04282=1066.988,328.440,-99.770,174.290,32.924,156.047
C04283=1066.981,328.192,-99.736,174.287,32.919,156.046
C04284=1066.975,327.944,-99.702,174.283,32.915,156.045
C04285=1066.968,327.697,-99.668,174.280,32.910,156.044
C04286=1066.962,327.449,-99.634,174.277,32.905,156.043
C04287=1066.956,327.202,-99.600,174.273,32.900,156.042
C04288=1066.949,326.954,-99.566,174.270,32.895,156.041
C04289=1066.943,326.707,-99.532,174.266,32.891,156.040
C04290=1066.936,326.459,-99.499,174.263,32.886,156.039
C04291=1066.930,326.212,-99.465,174.260,32.882,156.038
C04292=1066.923,325.964,-99.431,174.256,32.877,156.037
C04293=1066.917,325.717,-99.397,174.253,32.872,156.037
C04294=1066.910,325.469,-99.362,174.250,32.867,156.036
C04295=1066.904,325.221,-99.329,174.246,32.863,156.035
C04296=1066.898,324.973,-99.295,174.243,32.858,156.034
C04297=1066.891,324.726,-99.262,174.240,32.854,156.033
C04298=1066.886,324.478,-99.228,174.236,32.849,156.032
C04299=1066.878,324.230,-99.194,174.233,32.844,156.031
C04300=1066.872,323.983,-99.160,174.230,32.840,156.030
C04301=1066.866,323.735,-99.127,174.226,32.835,156.029
C04302=1066.860,323.488,-99.093,174.223,32.830,156.028
C04303=1066.854,323.240,-99.059,174.221,32.826,156.027
C04304=1066.847,322.992,-99.026,174.217,32.821,156.027
C04305=1066.841,322.745,-98.992,174.214,32.817,156.026
C04306=1066.834,322.496,-98.959,174.211,32.812,156.025
C04307=1066.828,322.249,-98.925,174.207,32.807,156.024
C04308=1066.822,322.002,-98.892,174.204,32.803,156.023
C04309=1066.816,321.754,-98.858,174.201,32.798,156.022
C04310=1066.809,321.506,-98.825,174.197,32.793,156.021
C04311=1066.803,321.259,-98.791,174.194,32.789,156.020
C04312=1066.797,321.011,-98.758,174.191,32.784,156.019
C04313=1066.791,320.763,-98.724,174.188,32.779,156.018
C04314=1066.784,320.516,-98.691,174.184,32.775,156.017
C04315=1066.779,320.268,-98.657,174.181,32.770,156.017
C04316=1066.772,320.020,-98.624,174.178,32.766,156.016
C04317=1066.766,319.772,-98.591,174.174,32.761,156.015
C04318=1066.759,319.525,-98.557,174.171,32.757,156.014
C04319=1066.754,319.277,-98.524,174.168,32.752,156.013
C04320=1066.747,319.029,-98.491,174.165,32.748,156.012
C04321=1066.741,318.782,-98.457,174.161,32.743,156.011
C04322=1066.736,318.548,-98.426,174.158,32.739,156.010
C04323=1066.730,318.315,-98.394,174.155,32.734,156.010
C04324=1066.724,318.081,-98.363,174.152,32.730,156.009
C04325=1066.718,317.848,-98.331,174.149,32.725,156.008
C04326=1066.712,317.615,-98.301,174.146,32.721,156.007
C04327=1066.707,317.381,-98.269,174.143,32.717,156.006
C04328=1066.701,317.148,-98.238,174.140,32.713,156.005
C04329=1066.695,316.915,-98.206,174.137,32.709,156.005
C04330=1066.688,316.667,-98.173,174.134,32.704,156.004
C04331=1066.682,316.419,-98.140,174.130,32.699,156.003
C04332=1066.676,316.171,-98.107,174.127,32.695,156.002
C04333=1066.671,315.923,-98.074,174.124,32.690,156.001
C04334=1066.664,315.676,-98.041,174.121,32.686,156.000
C04335=1066.659,315.428,-98.008,174.118,32.681,155.999
C04336=1066.652,315.180,-97.975,174.114,32.677,155.998
C04337=1066.646,314.933,-97.942,174.112,32.672,155.998
C04338=1066.640,314.685,-97.908,174.109,32.667,155.997
C04339=1066.634,314.438,-97.875,174.106,32.663,155.996
C04340=1066.628,314.190,-97.843,174.103,32.658,155.995
C04341=1066.622,313.942,-97.809,174.099,32.654,155.994
C04342=1066.615,313.694,-97.776,174.096,32.650,155.993
C04343=1066.609,313.446,-97.745,174.093,32.645,155.992
C04344=1066.602,313.198,-97.712,174.090,32.641,155.992
C04345=1066.596,312.951,-97.679,174.086,32.636,155.991
C04346=1066.590,312.703,-97.647,174.083,32.632,155.990
C04347=1066.583,312.456,-97.614,174.080,32.628,155.989
C04348=1066.577,312.207,-97.581,174.077,32.623,155.988
C04349=1066.570,311.960,-97.548,174.074,32.619,155.987
C04350=1066.564,311.712,-97.516,174.070,32.614,155.987
C04351=1066.558,311.464,-97.483,174.067,32.610,155.986
C04352=1066.552,311.216,-97.450,174.064,32.606,155.985
C04353=1066.545,310.969,-97.418,174.061,32.601,155.984
C04354=1066.539,310.721,-97.386,174.058,32.597,155.983
C04355=1066.532,310.473,-97.354,174.054,32.593,155.982
C04356=1066.526,310.226,-97.321,174.051,32.588,155.982
C04357=1066.520,309.978,-97.288,174.049,32.584,155.981
C04358=1066.514,309.730,-97.256,174.046,32.580,155.980
C04359=1066.507,309.482,-97.223,174.043,32.575,155.979
C04360=1066.501,309.235,-97.191,174.039,32.571,155.978
C04361=1066.495,308.987,-97.159,174.036,32.567,155.977
C04362=1066.488,308.739,-97.126,174.033,32.562,155.977
C04363=1066.482,308.491,-97.094,174.030,32.558,155.976
C04364=1066.476,308.243,-97.062,174.027,32.554,155.975
C04365=1066.470,307.996,-97.029,174.024,32.549,155.974
C04366=1066.464,307.748,-96.997,174.020,32.545,155.973
C04367=1066.457,307.500,-96.964,174.017,32.540,155.972
C04368=1066.451,307.252,-96.932,174.014,32.536,155.972
C04369=1066.444,307.005,-96.900,174.011,32.532,155.971
C04370=1066.438,306.756,-96.868,174.008,32.528,155.970
C04371=1066.432,306.509,-96.835,174.005,32.524,155.969
C04372=1066.426,306.260,-96.803,174.002,32.519,155.968
C04373=1066.420,306.014,-96.771,173.999,32.514,155.967
C04374=1066.414,305.766,-96.739,173.996,32.510,155.967
C04375=1066.407,305.518,-96.707,173.993,32.506,155.966
C04376=1066.401,305.270,-96.675,173.990,32.502,155.965
C04377=1066.395,305.022,-96.643,173.987,32.497,155.964
C04378=1066.390,304.790,-96.612,173.984,32.493,155.963
C04379=1066.383,304.558,-96.582,173.981,32.489,155.963
C04380=1066.378,304.327,-96.552,173.978,32.485,155.962
C04381=1066.372,304.096,-96.522,173.975,32.481,155.961
C04382=1066.366,303.864,-96.493,173.972,32.477,155.960
C04383=1066.360,303.632,-96.462,173.969,32.473,155.960
C04384=1066.355,303.401,-96.432,173.967,32.469,155.959
C04385=1066.349,303.169,-96.403,173.964,32.465,155.958
C04386=1066.343,302.922,-96.371,173.961,32.461,155.957
C04387=1066.337,302.673,-96.338,173.958,32.457,155.957
C04388=1066.331,302.426,-96.307,173.955,32.452,155.956
C04389=1066.325,302.178,-96.275,173.952,32.448,155.955
C04390=1066.318,301.930,-96.243,173.949,32.444,155.954
C04391=1066.312,301.682,-96.211,173.946,32.439,155.953
C04392=1066.307,301.435,-96.179,173.943,32.435,155.952
C04393=1066.300,301.187,-96.148,173.940,32.431,155.952
C04394=1066.294,300.939,-96.116,173.937,32.426,155.951
C04395=1066.288,300.690,-96.083,173.934,32.422,155.950
C04396=1066.283,300.443,-96.052,173.931,32.418,155.949
C04397=1066.276,300.196,-96.020,173.928,32.414,155.948
C04398=1066.270,299.947,-95.988,173.925,32.409,155.948
C04399=1066.264,299.700,-95.956,173.922,32.405,155.947
C04400=1066.258,299.452,-95.925,173.920,32.401,155.946
C04401=1066.252,299.204,-95.893,173.917,32.397,155.945
C04402=1066.246,298.956,-95.861,173.914,32.392,155.944
C04403=1066.240,298.708,-95.829,173.911,32.388,155.944
C04404=1066.234,298.460,-95.797,173.908,32.384,155.943
C04405=1066.228,298.213,-95.766,173.905,32.379,155.942
C04406=1066.222,297.964,-95.734,173.902,32.375,155.941
C04407=1066.216,297.717,-95.703,173.898,32.371,155.940
C04408=1066.210,297.469,-95.671,173.895,32.367,155.940
C04409=1066.204,297.221,-95.639,173.892,32.362,155.939
C04410=1066.198,296.973,-95.608,173.889,32.358,155.938
C04411=1066.192,296.725,-95.576,173.886,32.354,155.937
C04412=1066.186,296.477,-95.545,173.884,32.350,155.936
C04413=1066.180,296.230,-95.514,173.881,32.345,155.936
C04414=1066.174,295.981,-95.482,173.878,32.341,155.935
C04415=1066.167,295.733,-95.450,173.875,32.337,155.934
C04416=1066.162,295.485,-95.419,173.872,32.333,155.933
C04417=1066.155,295.237,-95.388,173.869,32.329,155.932
C04418=1066.149,294.990,-95.357,173.866,32.324,155.932
C04419=1066.143,294.742,-95.325,173.863,32.320,155.931
C04420=1066.137,294.493,-95.294,173.860,32.316,155.930
C04421=1066.130,294.246,-95.263,173.857,32.312,155.929
C04422=1066.124,293.998,-95.231,173.854,32.308,155.929
C04423=1066.118,293.750,-95.200,173.852,32.304,155.928
C04424=1066.112,293.502,-95.169,173.849,32.299,155.927
C04425=1066.106,293.254,-95.137,173.846,32.295,155.926
C04426=1066.100,293.006,-95.107,173.843,32.291,155.925
C04427=1066.093,292.758,-95.075,173.840,32.287,155.925
C04428=1066.087,292.510,-95.045,173.837,32.283,155.924
C04429=1066.082,292.262,-95.013,173.834,32.279,155.923
C04430=1066.075,292.014,-94.982,173.831,32.274,155.922
C04431=1066.069,291.767,-94.951,173.828,32.271,155.922
C04432=1066.063,291.518,-94.919,173.825,32.266,155.921
C04433=1066.057,291.271,-94.889,173.824,32.262,155.920
C04434=1066.051,291.047,-94.861,173.821,32.258,155.919
C04435=1066.046,290.823,-94.833,173.818,32.255,155.919
C04436=1066.040,290.598,-94.805,173.815,32.251,155.918
C04437=1066.034,290.374,-94.776,173.813,32.247,155.917
C04438=1066.029,290.150,-94.749,173.810,32.244,155.917
C04439=1066.024,289.926,-94.720,173.807,32.239,155.916
C04440=1066.018,289.702,-94.693,173.805,32.236,155.915
C04441=1066.012,289.478,-94.665,173.802,32.232,155.914
C04442=1066.007,289.230,-94.634,173.799,32.228,155.914
C04443=1066.000,288.982,-94.603,173.797,32.224,155.913
C04444=1065.995,288.734,-94.572,173.794,32.220,155.912
C04445=1065.988,288.485,-94.542,173.791,32.215,155.911
C04446=1065.982,288.238,-94.510,173.788,32.212,155.911
C04447=1065.976,287.990,-94.480,173.785,32.207,155.910
C04448=1065.970,287.742,-94.449,173.783,32.203,155.909
C04449=1065.963,287.493,-94.419,173.780,32.200,155.908
C04450=1065.957,287.246,-94.388,173.777,32.195,155.908
C04451=1065.951,286.998,-94.357,173.774,32.192,155.907
C04452=1065.945,286.750,-94.327,173.772,32.187,155.906
C04453=1065.939,286.501,-94.296,173.769,32.183,155.905
C04454=1065.933,286.254,-94.265,173.766,32.179,155.905
C04455=1065.926,286.006,-94.234,173.763,32.175,155.904
C04456=1065.920,285.758,-94.204,173.760,32.171,155.903
C04457=1065.914,285.510,-94.173,173.757,32.167,155.902
C04458=1065.908,285.261,-94.143,173.754,32.163,155.902
C04459=1065.902,285.014,-94.112,173.751,32.159,155.901
C04460=1065.896,284.765,-94.082,173.749,32.155,155.900
C04461=1065.890,284.517,-94.051,173.747,32.150,155.899
C04462=1065.884,284.270,-94.020,173.744,32.147,155.899
C04463=1065.877,284.022,-93.989,173.741,32.142,155.898
C04464=1065.872,283.774,-93.959,173.738,32.138,155.897
C04465=1065.866,283.526,-93.929,173.735,32.134,155.896
C04466=1065.859,283.277,-93.898,173.732,32.130,155.896
C04467=1065.854,283.030,-93.868,173.729,32.126,155.895
C04468=1065.846,282.781,-93.838,173.726,32.122,155.894
C04469=1065.841,282.534,-93.807,173.725,32.118,155.893
C04470=1065.835,282.286,-93.777,173.722,32.114,155.893
C04471=1065.828,282.037,-93.746,173.719,32.110,155.892
C04472=1065.823,281.789,-93.716,173.716,32.105,155.891
C04473=1065.817,281.541,-93.686,173.713,32.102,155.890
C04474=1065.811,281.293,-93.656,173.710,32.097,155.890
C04475=1065.805,281.045,-93.625,173.707,32.093,155.889
C04476=1065.799,280.797,-93.595,173.705,32.089,155.888
C04477=1065.793,280.549,-93.564,173.702,32.085,155.887
C04478=1065.787,280.300,-93.534,173.700,32.081,155.886
C04479=1065.780,280.053,-93.504,173.697,32.077,155.886
C04480=1065.775,279.804,-93.474,173.694,32.073,155.885
C04481=1065.769,279.557,-93.444,173.691,32.069,155.884
C04482=1065.762,279.308,-93.413,173.688,32.065,155.883
C04483=1065.756,279.061,-93.383,173.686,32.061,155.883
C04484=1065.750,278.812,-93.354,173.683,32.057,155.882
C04485=1065.744,278.564,-93.323,173.681,32.053,155.881
C04486=1065.737,278.316,-93.293,173.678,32.049,155.881
C04487=1065.732,278.068,-93.263,173.675,32.045,155.880
C04488=1065.726,277.820,-93.233,173.672,32.041,155.879
C04489=1065.720,277.571,-93.203,173.670,32.037,155.878
C04490=1065.714,277.353,-93.177,173.667,32.033,155.878
C04491=1065.709,277.134,-93.151,173.665,32.030,155.877
C04492=1065.703,276.915,-93.123,173.662,32.026,155.876
C04493=1065.698,276.697,-93.097,173.660,32.023,155.876
C04494=1065.693,276.477,-93.071,173.658,32.019,155.875
C04495=1065.688,276.258,-93.044,173.656,32.015,155.874
C04496=1065.682,276.040,-93.018,173.653,32.012,155.874
C04497=1065.676,275.821,-92.992,173.651,32.009,155.873
C04498=1065.671,275.573,-92.962,173.648,32.004,155.872
C04499=1065.665,275.325,-92.932,173.645,32.001,155.872
C04500=1065.658,275.076,-92.902,173.642,31.996,155.871
C04501=1065.652,274.828,-92.872,173.641,31.993,155.870
C04502=1065.646,274.580,-92.843,173.638,31.988,155.869
C04503=1065.640,274.332,-92.813,173.635,31.984,155.869
C04504=1065.635,274.084,-92.783,173.632,31.980,155.868
C04505=1065.628,273.836,-92.753,173.629,31.976,155.867
C04506=1065.622,273.587,-92.723,173.627,31.972,155.867
C04507=1065.616,273.340,-92.693,173.624,31.968,155.866
C04508=1065.610,273.091,-92.664,173.621,31.964,155.865
C04509=1065.604,272.843,-92.634,173.619,31.960,155.864
C04510=1065.598,272.595,-92.604,173.616,31.956,155.864
C04511=1065.592,272.347,-92.575,173.614,31.952,155.863
C04512=1065.586,272.099,-92.546,173.611,31.948,155.862
C04513=1065.579,271.850,-92.516,173.608,31.944,155.861
C04514=1065.574,271.602,-92.486,173.605,31.940,155.861
C04515=1065.567,271.354,-92.457,173.603,31.936,155.860
C04516=1065.561,271.106,-92.427,173.601,31.932,155.859
C04517=1065.555,270.858,-92.398,173.598,31.928,155.859
C04518=1065.550,270.609,-92.368,173.595,31.924,155.858
C04519=1065.543,270.361,-92.339,173.592,31.920,155.857
C04520=1065.537,270.114,-92.309,173.590,31.916,155.856
C04521=1065.531,269.865,-92.280,173.587,31.912,155.856
C04522=1065.525,269.617,-92.250,173.585,31.908,155.855
C04523=1065.520,269.369,-92.221,173.582,31.904,155.854
C04524=1065.513,269.120,-92.191,173.580,31.901,155.853
C04525=1065.506,268.872,-92.162,173.577,31.896,155.853
C04526=1065.501,268.624,-92.132,173.574,31.892,155.852
C04527=1065.494,268.376,-92.103,173.572,31.888,155.851
C04528=1065.488,268.128,-92.074,173.569,31.884,155.850
C04529=1065.483,267.879,-92.044,173.567,31.881,155.850
C04530=1065.476,267.631,-92.015,173.564,31.876,155.849
C04531=1065.470,267.383,-91.986,173.562,31.873,155.848
C04532=1065.464,267.135,-91.957,173.559,31.868,155.848
C04533=1065.458,266.887,-91.928,173.556,31.865,155.847
C04534=1065.452,266.638,-91.899,173.553,31.860,155.846
C04535=1065.446,266.390,-91.869,173.551,31.857,155.845
C04536=1065.440,266.142,-91.840,173.549,31.853,155.845
C04537=1065.434,265.894,-91.811,173.546,31.848,155.844
C04538=1065.428,265.646,-91.782,173.544,31.845,155.843
C04539=1065.422,265.397,-91.753,173.541,31.840,155.843
C04540=1065.416,265.149,-91.723,173.538,31.837,155.842
C04541=1065.410,264.901,-91.694,173.535,31.832,155.841
C04542=1065.404,264.653,-91.665,173.534,31.829,155.840
C04543=1065.397,264.405,-91.636,173.531,31.825,155.840
C04544=1065.392,264.156,-91.606,173.528,31.821,155.839
C04545=1065.386,263.908,-91.577,173.526,31.817,155.838
C04546=1065.381,263.690,-91.552,173.523,31.813,155.838
C04547=1065.375,263.474,-91.527,173.521,31.809,155.837
C04548=1065.370,263.257,-91.501,173.519,31.806,155.836
C04549=1065.364,263.040,-91.477,173.517,31.803,155.836
C04550=1065.359,262.823,-91.451,173.515,31.800,155.835
C04551=1065.353,262.606,-91.426,173.512,31.796,155.835
C04552=1065.348,262.389,-91.400,173.510,31.793,155.834
C04553=1065.342,262.171,-91.376,173.508,31.790,155.833
C04554=1065.336,261.923,-91.347,173.505,31.785,155.833
C04555=1065.330,261.675,-91.318,173.502,31.781,155.832
C04556=1065.324,261.426,-91.289,173.501,31.778,155.831
C04557=1065.317,261.178,-91.260,173.498,31.773,155.830
C04558=1065.311,260.930,-91.231,173.495,31.770,155.830
C04559=1065.305,260.681,-91.203,173.493,31.766,155.829
C04560=1065.299,260.433,-91.174,173.490,31.762,155.828
C04561=1065.293,260.186,-91.145,173.487,31.758,155.828
C04562=1065.287,259.937,-91.117,173.486,31.754,155.827
C04563=1065.281,259.689,-91.088,173.483,31.750,155.826
C04564=1065.274,259.441,-91.060,173.480,31.746,155.825
C04565=1065.268,259.192,-91.031,173.478,31.742,155.825
C04566=1065.262,258.944,-91.002,173.475,31.739,155.824
C04567=1065.256,258.696,-90.974,173.472,31.734,155.823
C04568=1065.250,258.447,-90.945,173.471,31.731,155.823
C04569=1065.244,258.199,-90.916,173.468,31.727,155.822
C04570=1065.238,257.951,-90.887,173.465,31.723,155.821
C04571=1065.232,257.702,-90.859,173.463,31.719,155.821
C04572=1065.225,257.455,-90.831,173.460,31.715,155.820
C04573=1065.219,257.206,-90.803,173.457,31.711,155.819
C04574=1065.213,256.958,-90.774,173.456,31.707,155.818
C04575=1065.207,256.709,-90.745,173.453,31.703,155.818
C04576=1065.201,256.461,-90.716,173.450,31.699,155.817
C04577=1065.195,256.213,-90.688,173.448,31.695,155.816
C04578=1065.189,255.965,-90.659,173.445,31.691,155.816
C04579=1065.183,255.716,-90.631,173.444,31.687,155.815
C04580=1065.177,255.468,-90.603,173.441,31.683,155.814
C04581=1065.170,255.219,-90.574,173.438,31.679,155.813
C04582=1065.165,254.971,-90.546,173.436,31.675,155.813
C04583=1065.159,254.723,-90.517,173.433,31.671,155.812
C04584=1065.153,254.474,-90.489,173.430,31.668,155.811
C04585=1065.146,254.226,-90.461,173.429,31.663,155.811
C04586=1065.140,253.978,-90.432,173.426,31.660,155.810
C04587=1065.135,253.730,-90.404,173.424,31.656,155.809
C04588=1065.129,253.481,-90.376,173.421,31.652,155.808
C04589=1065.123,253.232,-90.347,173.418,31.648,155.808
C04590=1065.117,252.985,-90.319,173.416,31.644,155.807
C04591=1065.110,252.736,-90.291,173.414,31.640,155.806
C04592=1065.104,252.488,-90.263,173.412,31.636,155.806
C04593=1065.098,252.239,-90.234,173.409,31.632,155.805
C04594=1065.093,251.992,-90.206,173.406,31.628,155.804
C04595=1065.087,251.743,-90.177,173.404,31.624,155.803
C04596=1065.080,251.494,-90.150,173.402,31.620,155.803
C04597=1065.075,251.246,-90.122,173.400,31.616,155.802
C04598=1065.069,250.998,-90.093,173.397,31.612,155.801
C04599=1065.063,250.749,-90.064,173.395,31.608,155.801
C04600=1065.057,250.502,-90.037,173.392,31.604,155.800
C04601=1065.051,250.253,-90.009,173.389,31.600,155.799
C04602=1065.046,250.035,-89.984,173.388,31.596,155.798
C04603=1065.040,249.816,-89.959,173.386,31.593,155.798
C04604=1065.035,249.599,-89.935,173.384,31.589,155.797
C04605=1065.030,249.380,-89.910,173.381,31.586,155.797
C04606=1065.025,249.162,-89.885,173.379,31.583,155.796
C04607=1065.020,248.943,-89.860,173.377,31.579,155.795
C04608=1065.014,248.726,-89.836,173.376,31.575,155.795
C04609=1065.009,248.507,-89.811,173.374,31.572,155.794
C04610=1065.004,248.259,-89.783,173.371,31.568,155.793
C04611=1064.998,248.010,-89.754,173.368,31.564,155.793
C04612=1064.992,247.763,-89.727,173.366,31.560,155.792
C04613=1064.986,247.514,-89.699,173.364,31.556,155.791
C04614=1064.980,247.265,-89.670,173.362,31.552,155.790
C04615=1064.974,247.017,-89.643,173.359,31.548,155.790
C04616=1064.968,246.769,-89.615,173.357,31.544,155.789
C04617=1064.962,246.521,-89.587,173.354,31.540,155.788
C04618=1064.956,246.272,-89.560,173.353,31.536,155.788
C04619=1064.951,246.024,-89.532,173.350,31.532,155.787
C04620=1064.944,245.775,-89.504,173.348,31.528,155.786
C04621=1064.938,245.526,-89.476,173.345,31.524,155.785
C04622=1064.932,245.279,-89.448,173.343,31.520,155.785
C04623=1064.926,245.030,-89.420,173.341,31.516,155.784
C04624=1064.920,244.782,-89.393,173.339,31.512,155.783
C04625=1064.914,244.533,-89.365,173.336,31.508,155.783
C04626=1064.908,244.285,-89.338,173.333,31.504,155.782
C04627=1064.902,244.036,-89.309,173.331,31.500,155.781
C04628=1064.895,243.788,-89.282,173.329,31.496,155.780
C04629=1064.890,243.540,-89.254,173.327,31.492,155.780
C04630=1064.884,243.291,-89.227,173.324,31.488,155.779
C04631=1064.878,243.043,-89.199,173.322,31.484,155.778
C04632=1064.872,242.794,-89.171,173.319,31.480,155.778
C04633=1064.866,242.546,-89.143,173.318,31.476,155.777
C04634=1064.860,242.297,-89.116,173.315,31.472,155.776
C04635=1064.855,242.049,-89.088,173.313,31.468,155.775
C04636=1064.848,241.801,-89.060,173.310,31.464,155.775
C04637=1064.842,241.552,-89.034,173.308,31.460,155.774
C04638=1064.836,241.304,-89.005,173.306,31.456,155.773
C04639=1064.831,241.055,-88.979,173.304,31.453,155.773
C04640=1064.824,240.807,-88.951,173.301,31.448,155.772
C04641=1064.818,240.559,-88.924,173.299,31.445,155.771
C04642=1064.812,240.310,-88.896,173.296,31.441,155.771
C04643=1064.806,240.062,-88.869,173.295,31.436,155.770
C04644=1064.800,239.813,-88.842,173.292,31.433,155.769
C04645=1064.794,239.565,-88.814,173.290,31.429,155.768
C04646=1064.788,239.316,-88.787,173.287,31.425,155.768
C04647=1064.782,239.068,-88.759,173.285,31.421,155.767
C04648=1064.775,238.819,-88.732,173.284,31.417,155.766
C04649=1064.769,238.571,-88.705,173.281,31.413,155.765
C04650=1064.764,238.322,-88.677,173.279,31.409,155.765
C04651=1064.758,238.074,-88.650,173.276,31.405,155.764
C04652=1064.751,237.825,-88.623,173.274,31.401,155.763
C04653=1064.745,237.577,-88.596,173.272,31.397,155.763
C04654=1064.739,237.328,-88.569,173.270,31.393,155.762
C04655=1064.734,237.080,-88.541,173.267,31.389,155.761
C04656=1064.727,236.831,-88.514,173.265,31.385,155.761
C04657=1064.721,236.583,-88.487,173.263,31.381,155.760
C04658=1064.715,236.362,-88.462,173.261,31.378,155.759
C04659=1064.711,236.141,-88.438,173.259,31.374,155.759
C04660=1064.705,235.919,-88.414,173.257,31.370,155.758
C04661=1064.700,235.698,-88.390,173.255,31.367,155.757
C04662=1064.695,235.476,-88.365,173.253,31.363,155.757
C04663=1064.689,235.255,-88.341,173.251,31.360,155.756
C04664=1064.684,235.034,-88.317,173.249,31.356,155.755
C04665=1064.678,234.812,-88.293,173.247,31.353,155.755
C04666=1064.673,234.564,-88.266,173.244,31.348,155.754
C04667=1064.667,234.316,-88.239,173.243,31.345,155.753
C04668=1064.660,234.067,-88.212,173.241,31.341,155.753
C04669=1064.655,233.819,-88.185,173.238,31.337,155.752
C04670=1064.649,233.570,-88.158,173.236,31.333,155.751
C04671=1064.642,233.322,-88.131,173.233,31.329,155.750
C04672=1064.636,233.073,-88.104,173.232,31.325,155.750
C04673=1064.630,232.824,-88.077,173.230,31.321,155.749
C04674=1064.624,232.576,-88.050,173.227,31.317,155.748
C04675=1064.619,232.328,-88.024,173.225,31.313,155.748
C04676=1064.613,232.078,-87.996,173.223,31.309,155.747
C04677=1064.607,231.831,-87.969,173.221,31.305,155.746
C04678=1064.601,231.582,-87.942,173.218,31.301,155.745
C04679=1064.595,231.333,-87.915,173.216,31.297,155.745
C04680=1064.589,231.085,-87.888,173.214,31.293,155.744
C04681=1064.583,230.836,-87.862,173.212,31.289,155.743
C04682=1064.577,230.588,-87.835,173.210,31.285,155.743
C04683=1064.571,230.339,-87.808,173.207,31.281,155.742
C04684=1064.565,230.091,-87.782,173.205,31.277,155.741
C04685=1064.559,229.842,-87.755,173.204,31.273,155.740
C04686=1064.552,229.594,-87.728,173.201,31.269,155.740
C04687=1064.546,229.346,-87.701,173.199,31.265,155.739
C04688=1064.541,229.097,-87.675,173.196,31.261,155.738
C04689=1064.534,228.848,-87.648,173.194,31.257,155.738
C04690=1064.529,228.599,-87.621,173.193,31.253,155.737
C04691=1064.523,228.351,-87.595,173.190,31.249,155.736
C04692=1064.516,228.103,-87.569,173.188,31.245,155.736
C04693=1064.510,227.854,-87.542,173.185,31.241,155.735
C04694=1064.504,227.606,-87.515,173.184,31.237,155.734
C04695=1064.498,227.357,-87.488,173.182,31.233,155.733
C04696=1064.493,227.109,-87.462,173.179,31.229,155.733
C04697=1064.486,226.860,-87.435,173.177,31.225,155.732
C04698=1064.480,226.612,-87.409,173.176,31.221,155.731
C04699=1064.474,226.363,-87.382,173.173,31.217,155.731
C04700=1064.468,226.115,-87.355,173.171,31.213,155.730
C04701=1064.461,225.866,-87.330,173.168,31.209,155.729
C04702=1064.456,225.617,-87.303,173.167,31.205,155.728
C04703=1064.450,225.369,-87.276,173.165,31.201,155.728
C04704=1064.444,225.121,-87.250,173.162,31.197,155.727
C04705=1064.438,224.872,-87.223,173.160,31.193,155.726
C04706=1064.431,224.623,-87.197,173.158,31.189,155.726
C04707=1064.426,224.374,-87.171,173.156,31.185,155.725
C04708=1064.420,224.126,-87.144,173.154,31.181,155.724
C04709=1064.414,223.878,-87.118,173.152,31.177,155.723
C04710=1064.408,223.630,-87.091,173.149,31.173,155.723
C04711=1064.402,223.381,-87.066,173.148,31.169,155.722
C04712=1064.396,223.132,-87.039,173.146,31.165,155.721
C04713=1064.390,222.883,-87.012,173.143,31.161,155.721
C04714=1064.385,222.658,-86.989,173.141,31.157,155.720
C04715=1064.379,222.432,-86.965,173.140,31.153,155.719
C04716=1064.374,222.207,-86.940,173.138,31.150,155.719
C04717=1064.369,221.982,-86.917,173.136,31.146,155.718
C04718=1064.363,221.756,-86.893,173.134,31.143,155.717
C04719=1064.358,221.531,-86.869,173.133,31.139,155.717
C04720=1064.352,221.306,-86.846,173.131,31.135,155.716
C04721=1064.346,221.080,-86.822,173.128,31.132,155.715
C04722=1064.341,220.832,-86.795,173.126,31.128,155.715
C04723=1064.334,220.583,-86.770,173.124,31.124,155.714
C04724=1064.329,220.335,-86.743,173.122,31.120,155.713
C04725=1064.322,220.087,-86.717,173.120,31.115,155.712
C04726=1064.317,219.838,-86.691,173.118,31.112,155.712
C04727=1064.310,219.590,-86.665,173.116,31.107,155.711
C04728=1064.304,219.340,-86.639,173.114,31.103,155.710
C04729=1064.298,219.092,-86.613,173.112,31.100,155.710
C04730=1064.292,218.843,-86.587,173.110,31.095,155.709
C04731=1064.286,218.595,-86.561,173.108,31.092,155.708
C04732=1064.280,218.346,-86.535,173.106,31.087,155.707
C04733=1064.274,218.098,-86.509,173.104,31.084,155.707
C04734=1064.268,217.849,-86.483,173.101,31.079,155.706
C04735=1064.262,217.601,-86.457,173.100,31.075,155.705
C04736=1064.256,217.352,-86.431,173.098,31.071,155.705
C04737=1064.250,217.103,-86.406,173.095,31.067,155.704
C04738=1064.243,216.855,-86.380,173.093,31.063,155.703
C04739=1064.238,216.606,-86.354,173.092,31.059,155.702
C04740=1064.231,216.358,-86.328,173.090,31.056,155.702
C04741=1064.225,216.109,-86.301,173.087,31.051,155.701
C04742=1064.219,215.860,-86.276,173.085,31.047,155.700
C04743=1064.213,215.612,-86.249,173.084,31.043,155.700
C04744=1064.207,215.363,-86.224,173.081,31.039,155.699
C04745=1064.202,215.114,-86.198,173.079,31.035,155.698
C04746=1064.195,214.866,-86.172,173.077,31.031,155.697
C04747=1064.190,214.617,-86.146,173.076,31.027,155.697
C04748=1064.184,214.368,-86.121,173.073,31.022,155.696
C04749=1064.178,214.121,-86.095,173.071,31.019,155.695
C04750=1064.172,213.872,-86.069,173.069,31.014,155.694
C04751=1064.166,213.623,-86.044,173.068,31.011,155.694
C04752=1064.161,213.374,-86.018,173.065,31.006,155.693
C04753=1064.154,213.126,-85.992,173.063,31.002,155.692
C04754=1064.148,212.878,-85.966,173.062,30.998,155.692
C04755=1064.142,212.629,-85.941,173.059,30.994,155.691
C04756=1064.136,212.380,-85.915,173.057,30.990,155.690
C04757=1064.130,212.131,-85.890,173.055,30.986,155.689
C04758=1064.124,211.883,-85.863,173.054,30.982,155.689
C04759=1064.118,211.634,-85.838,173.051,30.978,155.688
C04760=1064.112,211.386,-85.813,173.049,30.974,155.687
C04761=1064.106,211.137,-85.787,173.047,30.969,155.686
C04762=1064.100,210.888,-85.761,173.046,30.966,155.686
C04763=1064.094,210.639,-85.736,173.043,30.961,155.685
C04764=1064.088,210.391,-85.711,173.041,30.958,155.684
C04765=1064.082,210.142,-85.684,173.040,30.953,155.684
C04766=1064.076,209.894,-85.659,173.038,30.950,155.683
C04767=1064.069,209.645,-85.633,173.036,30.945,155.682
C04768=1064.064,209.397,-85.608,173.033,30.941,155.681
C04769=1064.058,209.148,-85.583,173.032,30.937,155.681
C04770=1064.052,208.925,-85.560,173.030,30.933,155.680
C04771=1064.047,208.702,-85.537,173.028,30.930,155.679
C04772=1064.041,208.479,-85.515,173.026,30.926,155.679
C04773=1064.036,208.256,-85.492,173.025,30.922,155.678
C04774=1064.031,208.033,-85.469,173.023,30.919,155.677
C04775=1064.025,207.810,-85.446,173.021,30.915,155.677
C04776=1064.020,207.587,-85.424,173.019,30.911,155.676
C04777=1064.014,207.364,-85.401,173.018,30.908,155.675
C04778=1063.990,206.317,-85.297,172.853,30.827,155.669
C04779=1063.984,206.068,-85.272,172.852,30.824,155.668
C04780=1063.978,205.820,-85.249,172.849,30.821,155.668
C04781=1063.972,205.571,-85.223,172.847,30.818,155.667
C04782=1063.967,205.323,-85.199,172.844,30.815,155.667
C04783=1063.961,205.073,-85.175,172.843,30.812,155.666
C04784=1063.956,204.825,-85.150,172.840,30.808,155.666
C04785=1063.950,204.575,-85.126,172.838,30.805,155.665
C04786=1063.943,204.328,-85.101,172.835,30.802,155.665
C04787=1063.937,204.079,-85.077,172.834,30.799,155.664
C04788=1063.932,203.830,-85.052,172.832,30.795,155.664
C04789=1063.926,203.581,-85.028,172.829,30.792,155.663
C04790=1063.921,203.332,-85.004,172.827,30.789,155.663
C04791=1063.914,203.084,-84.979,172.825,30.786,155.662
C04792=1063.909,202.835,-84.955,172.823,30.783,155.662
C04793=1063.903,202.587,-84.930,172.820,30.780,155.661
C04794=1063.898,202.337,-84.906,172.818,30.776,155.661
C04795=1063.892,202.089,-84.881,172.816,30.773,155.660
C04796=1063.886,201.840,-84.857,172.814,30.770,155.660
C04797=1063.880,201.591,-84.833,172.811,30.767,155.659
C04798=1063.874,201.342,-84.809,172.809,30.764,155.659
C04799=1063.868,201.094,-84.785,172.807,30.760,155.658
C04800=1063.862,200.845,-84.761,172.805,30.758,155.658
C04801=1063.856,200.596,-84.737,172.803,30.755,155.657
C04802=1063.850,200.347,-84.713,172.800,30.751,155.657
C04803=1063.844,200.098,-84.688,172.798,30.749,155.656
C04804=1063.838,199.850,-84.665,172.796,30.745,155.656
C04805=1063.833,199.601,-84.640,172.794,30.742,155.655
C04806=1063.826,199.353,-84.616,172.791,30.739,155.655
C04807=1063.821,199.103,-84.592,172.789,30.736,155.654
C04808=1063.815,198.855,-84.568,172.788,30.733,155.654
C04809=1063.809,198.606,-84.543,172.785,30.730,155.653
C04810=1063.803,198.357,-84.520,172.783,30.727,155.653
C04811=1063.797,198.109,-84.496,172.780,30.723,155.652
C04812=1063.791,197.859,-84.472,172.779,30.721,155.652
C04813=1063.786,197.611,-84.448,172.776,30.717,155.651
C04814=1063.780,197.362,-84.424,172.774,30.714,155.651
C04815=1063.774,197.113,-84.400,172.772,30.712,155.650
C04816=1063.768,196.865,-84.376,172.770,30.708,155.650
C04817=1063.762,196.616,-84.351,172.768,30.705,155.649
C04818=1063.756,196.367,-84.328,172.765,30.702,155.649
C04819=1063.751,196.118,-84.304,172.763,30.699,155.648
C04820=1063.744,195.869,-84.280,172.762,30.696,155.648
C04821=1063.739,195.620,-84.256,172.759,30.693,155.647
C04822=1063.733,195.372,-84.232,172.757,30.690,155.647
C04823=1063.727,195.123,-84.208,172.754,30.686,155.646
C04824=1063.721,194.874,-84.185,172.753,30.684,155.646
C04825=1063.716,194.625,-84.160,172.751,30.681,155.645
C04826=1063.710,194.377,-84.137,172.748,30.677,155.645
C04827=1063.704,194.128,-84.113,172.746,30.675,155.644
C04828=1063.698,193.879,-84.089,172.744,30.671,155.644
C04829=1063.692,193.631,-84.066,172.742,30.668,155.643
C04830=1063.686,193.381,-84.041,172.740,30.665,155.643
C04831=1063.681,193.133,-84.018,172.737,30.662,155.642
C04832=1063.675,192.884,-83.994,172.736,30.659,155.642
C04833=1063.669,192.636,-83.970,172.734,30.656,155.642
C04834=1063.664,192.386,-83.946,172.731,30.653,155.641
C04835=1063.658,192.137,-83.922,172.729,30.650,155.641
C04836=1063.652,191.889,-83.900,172.727,30.647,155.640
C04837=1063.647,191.640,-83.875,172.725,30.644,155.640
C04838=1063.640,191.391,-83.851,172.723,30.641,155.639
C04839=1063.634,191.108,-83.825,172.720,30.637,155.638
C04840=1063.627,190.825,-83.798,172.718,30.634,155.638
C04841=1063.621,190.542,-83.771,172.716,30.630,155.637
C04842=1063.615,190.258,-83.744,172.713,30.626,155.637
C04843=1063.609,190.010,-83.720,172.711,30.624,155.636
C04844=1063.603,189.761,-83.697,172.709,30.620,155.636
C04845=1063.597,189.512,-83.673,172.707,30.618,155.635
C04846=1063.592,189.264,-83.650,172.705,30.615,155.635
C04847=1063.586,189.015,-83.626,172.702,30.611,155.634
C04848=1063.580,188.765,-83.602,172.701,30.609,155.634
C04849=1063.574,188.517,-83.579,172.699,30.605,155.633
C04850=1063.569,188.268,-83.555,172.696,30.602,155.633
C04851=1063.563,188.020,-83.531,172.694,30.599,155.633
C04852=1063.557,187.771,-83.508,172.693,30.596,155.632
C04853=1063.552,187.522,-83.484,172.690,30.593,155.631
C04854=1063.546,187.273,-83.461,172.688,30.590,155.631
C04855=1063.540,187.024,-83.437,172.686,30.587,155.630
C04856=1063.535,186.775,-83.414,172.684,30.584,155.630
C04857=1063.529,186.526,-83.391,172.682,30.581,155.630
C04858=1063.524,186.278,-83.366,172.680,30.578,155.629
C04859=1063.518,186.029,-83.343,172.677,30.575,155.629
C04860=1063.512,185.780,-83.320,172.676,30.572,155.628
C04861=1063.507,185.531,-83.296,172.674,30.568,155.628
C04862=1063.501,185.282,-83.273,172.672,30.566,155.627
C04863=1063.495,185.034,-83.250,172.669,30.562,155.627
C04864=1063.490,184.785,-83.226,172.668,30.560,155.626
C04865=1063.484,184.536,-83.203,172.666,30.557,155.626
C04866=1063.478,184.286,-83.180,172.663,30.554,155.625
C04867=1063.472,184.038,-83.156,172.661,30.550,155.625
C04868=1063.466,183.789,-83.133,172.660,30.548,155.624
C04869=1063.461,183.540,-83.110,172.657,30.545,155.624
C04870=1063.454,183.292,-83.088,172.655,30.542,155.623
C04871=1063.447,183.043,-83.064,172.653,30.539,155.623
C04872=1063.442,182.794,-83.041,172.652,30.537,155.623
C04873=1063.436,182.545,-83.018,172.649,30.533,155.622
C04874=1063.430,182.296,-82.995,172.647,30.530,155.622
C04875=1063.425,182.047,-82.972,172.645,30.528,155.621
C04876=1063.419,181.798,-82.949,172.643,30.524,155.621
C04877=1063.412,181.549,-82.925,172.641,30.522,155.620
C04878=1063.406,181.300,-82.902,172.639,30.519,155.620
C04879=1063.400,181.052,-82.880,172.636,30.516,155.619
C04880=1063.394,180.803,-82.857,172.635,30.513,155.619
C04881=1063.388,180.554,-82.834,172.633,30.510,155.618
C04882=1063.383,180.305,-82.811,172.631,30.507,155.618
C04883=1063.377,180.056,-82.788,172.628,30.504,155.618
C04884=1063.371,179.807,-82.765,172.627,30.501,155.617
C04885=1063.366,179.558,-82.742,172.625,30.499,155.617
C04886=1063.359,179.310,-82.720,172.623,30.496,155.616
C04887=1063.353,179.060,-82.697,172.620,30.492,155.616
C04888=1063.347,178.812,-82.673,172.619,30.490,155.615
C04889=1063.341,178.563,-82.650,172.617,30.487,155.615
C04890=1063.335,178.314,-82.627,172.614,30.484,155.614
C04891=1063.330,178.065,-82.604,172.612,30.481,155.614
C04892=1063.323,177.817,-82.582,172.611,30.478,155.614
C04893=1063.317,177.568,-82.559,172.609,30.475,155.613
C04894=1063.312,177.318,-82.537,172.606,30.472,155.613
C04895=1063.306,177.069,-82.514,172.604,30.470,155.612
C04896=1063.300,176.820,-82.491,172.603,30.467,155.612
C04897=1063.295,176.571,-82.468,172.601,30.464,155.611
C04898=1063.288,176.323,-82.445,172.598,30.461,155.611
C04899=1063.283,176.074,-82.422,172.596,30.458,155.610
C04900=1063.277,175.825,-82.399,172.595,30.455,155.610
C04901=1063.271,175.576,-82.376,172.593,30.453,155.609
C04902=1063.265,175.327,-82.354,172.591,30.449,155.609
C04903=1063.259,175.044,-82.328,172.588,30.446,155.608
C04904=1063.252,174.760,-82.302,172.586,30.442,155.608
C04905=1063.245,174.477,-82.276,172.584,30.439,155.607
C04906=1063.238,174.194,-82.250,172.581,30.436,155.607
C04907=1063.233,173.944,-82.228,172.580,30.433,155.606
C04908=1063.227,173.695,-82.205,172.578,30.431,155.606
C04909=1063.221,173.446,-82.182,172.576,30.427,155.605
C04910=1063.215,173.198,-82.159,172.573,30.424,155.605
C04911=1063.209,172.949,-82.137,172.572,30.422,155.605
C04912=1063.204,172.700,-82.115,172.570,30.419,155.604
C04913=1063.198,172.451,-82.092,172.568,30.416,155.604
C04914=1063.193,172.202,-82.069,172.566,30.413,155.603
C04915=1063.186,171.954,-82.047,172.564,30.410,155.603
C04916=1063.180,171.705,-82.024,172.562,30.407,155.602
C04917=1063.175,171.455,-82.002,172.560,30.405,155.602
C04918=1063.169,171.207,-81.979,172.558,30.401,155.601
C04919=1063.163,170.958,-81.956,172.557,30.399,155.601
C04920=1063.157,170.708,-81.934,172.554,30.396,155.601
C04921=1063.152,170.459,-81.911,172.552,30.393,155.600
C04922=1063.146,170.211,-81.889,172.550,30.390,155.600
C04923=1063.140,169.963,-81.866,172.549,30.387,155.599
C04924=1063.135,169.713,-81.844,172.547,30.384,155.599
C04925=1063.129,169.464,-81.821,172.545,30.381,155.598
C04926=1063.123,169.215,-81.799,172.543,30.378,155.598
C04927=1063.117,168.966,-81.777,172.541,30.375,155.597
C04928=1063.111,168.717,-81.754,172.539,30.373,155.597
C04929=1063.106,168.468,-81.732,172.537,30.369,155.596
C04930=1063.101,168.220,-81.709,172.536,30.367,155.596
C04931=1063.094,167.971,-81.686,172.533,30.364,155.596
C04932=1063.089,167.721,-81.664,172.531,30.361,155.595
C04933=1063.083,167.473,-81.641,172.529,30.358,155.595
C04934=1063.077,167.224,-81.620,172.528,30.355,155.594
C04935=1063.072,166.975,-81.597,172.526,30.352,155.594
C04936=1063.066,166.726,-81.575,172.524,30.349,155.593
C04937=1063.061,166.477,-81.552,172.522,30.346,155.593
C04938=1063.054,166.228,-81.529,172.520,30.343,155.592
C04939=1063.049,165.979,-81.508,172.518,30.341,155.592
C04940=1063.044,165.730,-81.485,172.516,30.337,155.591
C04941=1063.037,165.481,-81.463,172.514,30.335,155.591
C04942=1063.032,165.232,-81.440,172.513,30.332,155.591
C04943=1063.027,164.984,-81.418,172.511,30.329,155.590
C04944=1063.020,164.735,-81.396,172.508,30.326,155.590
C04945=1063.015,164.485,-81.374,172.506,30.323,155.589
C04946=1063.010,164.236,-81.351,172.505,30.320,155.589
C04947=1063.004,163.988,-81.329,172.503,30.318,155.588
C04948=1062.998,163.739,-81.307,172.501,30.314,155.588
C04949=1062.992,163.490,-81.284,172.499,30.312,155.587
C04950=1062.987,163.241,-81.263,172.498,30.309,155.587
C04951=1062.981,162.992,-81.240,172.496,30.306,155.586
C04952=1062.976,162.743,-81.218,172.493,30.303,155.586
C04953=1062.970,162.494,-81.197,172.492,30.300,155.586
C04954=1062.964,162.245,-81.174,172.490,30.297,155.585
C04955=1062.959,161.996,-81.151,172.488,30.294,155.585
C04956=1062.953,161.748,-81.129,172.486,30.291,155.584
C04957=1062.948,161.498,-81.107,172.485,30.288,155.584
C04958=1062.942,161.249,-81.085,172.483,30.286,155.583
C04959=1062.936,161.000,-81.063,172.481,30.282,155.583
C04960=1062.931,160.752,-81.041,172.478,30.280,155.582
C04961=1062.925,160.502,-81.019,172.477,30.277,155.582
C04962=1062.919,160.253,-80.997,172.475,30.274,155.582
C04963=1062.912,160.005,-80.975,172.473,30.271,155.581
C04964=1062.907,159.756,-80.953,172.471,30.268,155.581
C04965=1062.901,159.506,-80.932,172.470,30.266,155.580
C04966=1062.895,159.257,-80.910,172.468,30.263,155.580
C04967=1062.889,158.974,-80.885,172.465,30.260,155.579
C04968=1062.883,158.690,-80.859,172.464,30.256,155.579
C04969=1062.876,158.406,-80.835,172.461,30.253,155.578
C04970=1062.870,158.122,-80.810,172.459,30.250,155.578
C04971=1062.863,157.873,-80.788,172.457,30.248,155.577
C04972=1062.857,157.624,-80.766,172.456,30.244,155.577
C04973=1062.851,157.376,-80.745,172.454,30.242,155.576
C04974=1062.846,157.126,-80.723,172.452,30.239,155.576
C04975=1062.840,156.877,-80.701,172.450,30.236,155.576
C04976=1062.834,156.628,-80.680,172.448,30.233,155.575
C04977=1062.829,156.379,-80.657,172.446,30.230,155.575
C04978=1062.822,156.130,-80.635,172.444,30.228,155.574
C04979=1062.817,155.882,-80.614,172.443,30.225,155.574
C04980=1062.811,155.633,-80.592,172.441,30.222,155.573
C04981=1062.805,155.383,-80.570,172.439,30.219,155.573
C04982=1062.800,155.135,-80.549,172.437,30.216,155.573
C04983=1062.793,154.885,-80.527,172.436,30.214,155.572
C04984=1062.787,154.636,-80.505,172.434,30.211,155.572
C04985=1062.782,154.388,-80.484,172.432,30.208,155.571
C04986=1062.776,154.138,-80.462,172.430,30.206,155.571
C04987=1062.770,153.889,-80.440,172.428,30.203,155.571
C04988=1062.765,153.641,-80.419,172.426,30.199,155.570
C04989=1062.758,153.391,-80.397,172.424,30.197,155.570
C04990=1062.752,153.142,-80.376,172.422,30.194,155.569
C04991=1062.747,152.894,-80.354,172.421,30.191,155.569
C04992=1062.741,152.644,-80.332,172.419,30.189,155.568
C04993=1062.736,152.396,-80.311,172.417,30.186,155.568
C04994=1062.730,152.146,-80.289,172.416,30.183,155.567
C04995=1062.723,151.897,-80.268,172.414,30.180,155.567
C04996=1062.718,151.649,-80.246,172.412,30.177,155.567
C04997=1062.712,151.399,-80.225,172.410,30.175,155.566
C04998=1062.706,151.151,-80.203,172.409,30.172,155.566
C04999=1062.700,150.902,-80.182,172.407,30.169,155.565
C05000=1062.694,150.652,-80.160,172.405,30.166,155.565
C05001=1062.689,150.403,-80.139,172.402,30.163,155.564
C05002=1062.683,150.154,-80.117,172.401,30.161,155.564
C05003=1062.677,149.905,-80.096,172.399,30.158,155.564
C05004=1062.671,149.656,-80.075,172.397,30.155,155.563
C05005=1062.666,149.408,-80.053,172.395,30.153,155.563
C05006=1062.660,149.158,-80.032,172.394,30.150,155.562
C05007=1062.654,148.909,-80.011,172.392,30.147,155.562
C05008=1062.648,148.660,-79.989,172.390,30.144,155.561
C05009=1062.642,148.411,-79.968,172.389,30.141,155.561
C05010=1062.636,148.162,-79.947,172.387,30.139,155.561
C05011=1062.630,147.913,-79.925,172.385,30.136,155.560
C05012=1062.625,147.664,-79.904,172.383,30.133,155.560
C05013=1062.619,147.415,-79.883,172.382,30.131,155.559
C05014=1062.613,147.166,-79.861,172.380,30.128,155.559
C05015=1062.607,146.917,-79.840,172.378,30.125,155.559
C05016=1062.601,146.667,-79.819,172.376,30.122,155.558
C05017=1062.596,146.419,-79.798,172.375,30.119,155.558
C05018=1062.590,146.170,-79.776,172.373,30.117,155.557
C05019=1062.584,145.921,-79.755,172.371,30.114,155.557
C05020=1062.577,145.672,-79.734,172.369,30.111,155.556
C05021=1062.572,145.423,-79.713,172.368,30.109,155.556
C05022=1062.566,145.174,-79.691,172.366,30.106,155.556
C05023=1062.560,144.925,-79.671,172.363,30.103,155.555
C05024=1062.554,144.676,-79.649,172.362,30.100,155.555
C05025=1062.549,144.427,-79.628,172.360,30.098,155.554
C05026=1062.543,144.177,-79.607,172.358,30.095,155.554
C05027=1062.537,143.929,-79.586,172.356,30.092,155.553
C05028=1062.530,143.680,-79.565,172.355,30.089,155.553
C05029=1062.525,143.431,-79.544,172.353,30.086,155.553
C05030=1062.519,143.182,-79.523,172.351,30.084,155.552
C05031=1062.512,142.897,-79.499,172.349,30.080,155.552
C05032=1062.506,142.613,-79.475,172.348,30.078,155.551
C05033=1062.500,142.329,-79.450,172.345,30.074,155.551
C05034=1062.493,142.045,-79.426,172.343,30.071,155.550
C05035=1062.487,141.796,-79.406,172.342,30.068,155.550
C05036=1062.481,141.547,-79.384,172.340,30.066,155.549
C05037=1062.475,141.298,-79.364,172.338,30.063,155.549
C05038=1062.470,141.049,-79.343,172.336,30.060,155.549
C05039=1062.464,140.800,-79.322,172.335,30.057,155.548
C05040=1062.458,140.551,-79.300,172.333,30.055,155.548
C05041=1062.453,140.301,-79.279,172.331,30.052,155.547
C05042=1062.446,140.053,-79.259,172.330,30.049,155.547
C05043=1062.440,139.803,-79.238,172.328,30.046,155.546
C05044=1062.435,139.555,-79.217,172.326,30.043,155.546
C05045=1062.428,139.305,-79.196,172.324,30.041,155.546
C05046=1062.423,139.057,-79.175,172.323,30.038,155.545
C05047=1062.417,138.808,-79.154,172.321,30.035,155.545
C05048=1062.412,138.558,-79.134,172.319,30.033,155.544
C05049=1062.405,138.310,-79.113,172.317,30.030,155.544
C05050=1062.399,138.060,-79.092,172.316,30.027,155.543
C05051=1062.394,137.811,-79.071,172.314,30.025,155.543
C05052=1062.388,137.562,-79.051,172.312,30.022,155.543
C05053=1062.382,137.313,-79.030,172.311,30.019,155.542
C05054=1062.376,137.064,-79.009,172.309,30.017,155.542
C05055=1062.370,136.815,-78.988,172.307,30.014,155.541
C05056=1062.365,136.565,-78.968,172.305,30.011,155.541
C05057=1062.358,136.317,-78.947,172.304,30.008,155.541
C05058=1062.352,136.067,-78.926,172.302,30.006,155.540
C05059=1062.347,135.818,-78.905,172.300,30.003,155.540
C05060=1062.340,135.569,-78.884,172.298,30.000,155.539
C05061=1062.335,135.320,-78.864,172.297,29.998,155.539
C05062=1062.330,135.071,-78.843,172.295,29.994,155.538
C05063=1062.323,134.822,-78.822,172.293,29.992,155.538
C05064=1062.318,134.573,-78.802,172.292,29.989,155.538
C05065=1062.312,134.324,-78.782,172.290,29.986,155.537
C05066=1062.306,134.074,-78.761,172.288,29.984,155.537
C05067=1062.300,133.826,-78.740,172.286,29.981,155.536
C05068=1062.294,133.577,-78.720,172.285,29.978,155.536
C05069=1062.288,133.327,-78.699,172.284,29.976,155.536
C05070=1062.282,133.079,-78.679,172.282,29.973,155.535
C05071=1062.277,132.830,-78.657,172.280,29.970,155.535
C05072=1062.271,132.580,-78.637,172.279,29.968,155.534
C05073=1062.265,132.331,-78.617,172.277,29.965,155.534
C05074=1062.260,132.082,-78.596,172.275,29.962,155.534
C05075=1062.253,131.833,-78.576,172.274,29.960,155.533
C05076=1062.248,131.584,-78.554,172.272,29.957,155.533
C05077=1062.242,131.335,-78.534,172.270,29.954,155.532
C05078=1062.235,131.086,-78.514,172.268,29.951,155.532
C05079=1062.230,130.837,-78.494,172.267,29.949,155.531
C05080=1062.224,130.588,-78.474,172.265,29.946,155.531
C05081=1062.217,130.338,-78.453,172.263,29.943,155.531
C05082=1062.212,130.089,-78.433,172.262,29.941,155.530
C05083=1062.206,129.841,-78.413,172.260,29.938,155.530
C05084=1062.199,129.592,-78.392,172.258,29.935,155.529
C05085=1062.194,129.343,-78.371,172.256,29.933,155.529
C05086=1062.188,129.094,-78.351,172.255,29.930,155.529
C05087=1062.181,128.844,-78.331,172.253,29.927,155.528
C05088=1062.176,128.595,-78.310,172.251,29.924,155.528
C05089=1062.170,128.346,-78.290,172.249,29.922,155.527
C05090=1062.163,128.097,-78.270,172.248,29.920,155.527
C05091=1062.158,127.848,-78.250,172.246,29.917,155.527
C05092=1062.152,127.599,-78.230,172.244,29.914,155.526
C05093=1062.145,127.349,-78.209,172.243,29.912,155.526
C05094=1062.140,127.100,-78.189,172.242,29.909,155.525
C05095=1062.133,126.816,-78.166,172.239,29.906,155.525
C05096=1062.126,126.531,-78.143,172.237,29.903,155.525
C05097=1062.120,126.247,-78.120,172.236,29.900,155.524
C05098=1062.113,125.964,-78.097,172.234,29.897,155.524
C05099=1062.107,125.715,-78.076,172.232,29.894,155.523
C05100=1062.101,125.465,-78.056,172.231,29.891,155.523
C05101=1062.095,125.216,-78.036,172.229,29.889,155.522
C05102=1062.090,124.967,-78.016,172.227,29.886,155.522
C05103=1062.084,124.718,-77.996,172.225,29.883,155.522
C05104=1062.077,124.468,-77.976,172.224,29.881,155.521
C05105=1062.071,124.219,-77.956,172.222,29.878,155.521
C05106=1062.066,123.970,-77.936,172.220,29.875,155.520
C05107=1062.060,123.721,-77.916,172.219,29.873,155.520
C05108=1062.053,123.472,-77.895,172.217,29.870,155.520
C05109=1062.047,123.223,-77.875,172.216,29.867,155.519
C05110=1062.042,122.973,-77.855,172.214,29.865,155.519
C05111=1062.036,122.725,-77.835,172.213,29.862,155.518
C05112=1062.030,122.476,-77.816,172.211,29.859,155.518
C05113=1062.024,122.227,-77.796,172.209,29.857,155.517
C05114=1062.019,121.977,-77.775,172.208,29.854,155.517
C05115=1062.013,121.728,-77.755,172.206,29.851,155.517
C05116=1062.007,121.479,-77.735,172.204,29.848,155.516
C05117=1062.001,121.230,-77.715,172.202,29.846,155.516
C05118=1061.996,120.981,-77.695,172.201,29.843,155.515
C05119=1061.990,120.732,-77.675,172.199,29.840,155.515
C05120=1061.983,120.483,-77.655,172.197,29.838,155.515
C05121=1061.977,120.233,-77.635,172.197,29.835,155.514
C05122=1061.972,119.984,-77.615,172.195,29.832,155.514
C05123=1061.966,119.735,-77.595,172.193,29.830,155.513
C05124=1061.960,119.486,-77.575,172.191,29.826,155.513
C05125=1061.954,119.237,-77.556,172.190,29.824,155.512
C05126=1061.948,118.988,-77.536,172.188,29.821,155.512
C05127=1061.943,118.739,-77.515,172.186,29.818,155.512
C05128=1061.937,118.489,-77.496,172.185,29.816,155.511
C05129=1061.931,118.240,-77.476,172.183,29.813,155.511
C05130=1061.925,117.991,-77.456,172.181,29.810,155.510
C05131=1061.920,117.742,-77.436,172.180,29.808,155.510
C05132=1061.914,117.493,-77.416,172.179,29.805,155.510
C05133=1061.908,117.244,-77.396,172.177,29.802,155.509
C05134=1061.902,116.994,-77.377,172.175,29.799,155.509
C05135=1061.896,116.746,-77.357,172.174,29.797,155.508
C05136=1061.891,116.497,-77.336,172.172,29.794,155.508
C05137=1061.885,116.247,-77.317,172.170,29.791,155.508
C05138=1061.879,115.998,-77.297,172.168,29.789,155.507
C05139=1061.873,115.749,-77.277,172.167,29.786,155.507
C05140=1061.868,115.500,-77.258,172.166,29.783,155.506
C05141=1061.862,115.251,-77.238,172.164,29.781,155.506
C05142=1061.856,115.001,-77.218,172.163,29.778,155.505
C05143=1061.850,114.752,-77.198,172.161,29.775,155.505
C05144=1061.844,114.503,-77.178,172.159,29.772,155.505
C05145=1061.838,114.254,-77.158,172.158,29.769,155.504
C05146=1061.832,114.005,-77.138,172.156,29.767,155.504
C05147=1061.827,113.755,-77.119,172.154,29.764,155.503
C05148=1061.821,113.507,-77.099,172.153,29.761,155.503
C05149=1061.815,113.257,-77.080,172.152,29.759,155.502
C05150=1061.809,113.008,-77.060,172.150,29.756,155.502
C05151=1061.803,112.759,-77.041,172.148,29.754,155.502
C05152=1061.797,112.510,-77.021,172.146,29.751,155.501
C05153=1061.792,112.261,-77.002,172.145,29.748,155.501
C05154=1061.786,112.012,-76.982,172.143,29.746,155.501
C05155=1061.780,111.763,-76.962,172.141,29.743,155.500
C05156=1061.774,111.513,-76.943,172.140,29.740,155.500
C05157=1061.768,111.264,-76.923,172.139,29.738,155.499
C05158=1061.763,111.015,-76.904,172.137,29.735,155.499
C05159=1061.756,110.730,-76.881,172.136,29.732,155.498
C05160=1061.749,110.445,-76.859,172.133,29.729,155.498
C05161=1061.741,110.162,-76.838,172.131,29.725,155.497
C05162=1061.735,109.877,-76.816,172.130,29.723,155.497
C05163=1061.729,109.628,-76.796,172.128,29.720,155.497
C05164=1061.723,109.379,-76.776,172.126,29.717,155.496
C05165=1061.717,109.129,-76.757,172.125,29.715,155.496
C05166=1061.711,108.881,-76.737,172.124,29.712,155.495
C05167=1061.705,108.632,-76.719,172.122,29.709,155.495
C05168=1061.699,108.382,-76.699,172.120,29.707,155.495
C05169=1061.693,108.133,-76.679,172.119,29.704,155.494
C05170=1061.687,107.884,-76.660,172.117,29.702,155.494
C05171=1061.682,107.634,-76.641,172.115,29.699,155.494
C05172=1061.675,107.386,-76.621,172.113,29.696,155.493
C05173=1061.669,107.136,-76.602,172.113,29.694,155.493
C05174=1061.664,106.887,-76.583,172.111,29.691,155.492
C05175=1061.658,106.638,-76.563,172.109,29.688,155.492
C05176=1061.652,106.389,-76.544,172.108,29.686,155.491
C05177=1061.646,106.140,-76.525,172.106,29.683,155.491
C05178=1061.640,105.890,-76.506,172.104,29.680,155.491
C05179=1061.634,105.641,-76.486,172.103,29.677,155.490
C05180=1061.628,105.392,-76.467,172.102,29.675,155.490
C05181=1061.622,105.143,-76.448,172.100,29.672,155.489
C05182=1061.616,104.893,-76.429,172.098,29.669,155.489
C05183=1061.610,104.644,-76.410,172.097,29.667,155.489
C05184=1061.604,104.395,-76.390,172.095,29.664,155.488
C05185=1061.599,104.147,-76.371,172.093,29.661,155.488
C05186=1061.593,103.897,-76.352,172.092,29.659,155.488
C05187=1061.587,103.648,-76.333,172.091,29.657,155.487
C05188=1061.581,103.398,-76.314,172.089,29.654,155.487
C05189=1061.575,103.150,-76.294,172.087,29.651,155.486
C05190=1061.569,102.901,-76.275,172.086,29.648,155.486
C05191=1061.563,102.651,-76.256,172.084,29.646,155.485
C05192=1061.558,102.402,-76.236,172.082,29.643,155.485
C05193=1061.551,102.153,-76.218,172.081,29.640,155.485
C05194=1061.546,101.903,-76.199,172.080,29.638,155.484
C05195=1061.540,101.654,-76.179,172.078,29.635,155.484
C05196=1061.535,101.405,-76.160,172.077,29.632,155.483
C05197=1061.528,101.156,-76.142,172.075,29.630,155.483
C05198=1061.522,100.907,-76.122,172.073,29.627,155.483
C05199=1061.517,100.658,-76.103,172.071,29.624,155.482
C05200=1061.510,100.408,-76.084,172.071,29.622,155.482
C05201=1061.505,100.159,-76.065,172.069,29.619,155.481
C05202=1061.498,99.910,-76.046,172.067,29.616,155.481
C05203=1061.492,99.660,-76.027,172.066,29.613,155.481
C05204=1061.486,99.411,-76.008,172.064,29.611,155.480
C05205=1061.480,99.162,-75.989,172.062,29.609,155.480
C05206=1061.474,98.913,-75.970,172.061,29.606,155.479
C05207=1061.469,98.664,-75.951,172.060,29.603,155.479
C05208=1061.462,98.415,-75.933,172.058,29.601,155.479
C05209=1061.457,98.166,-75.914,172.056,29.598,155.478
C05210=1061.450,97.916,-75.895,172.055,29.595,155.478
C05211=1061.445,97.667,-75.876,172.053,29.592,155.477
C05212=1061.438,97.418,-75.857,172.051,29.590,155.477
C05213=1061.433,97.168,-75.838,172.051,29.588,155.477
C05214=1061.426,96.919,-75.820,172.049,29.585,155.476
C05215=1061.421,96.670,-75.801,172.047,29.582,155.476
C05216=1061.415,96.421,-75.782,172.045,29.580,155.476
C05217=1061.409,96.171,-75.763,172.044,29.577,155.475
C05218=1061.403,95.922,-75.744,172.042,29.574,155.475
C05219=1061.397,95.673,-75.725,172.041,29.572,155.474
C05220=1061.391,95.424,-75.707,172.040,29.569,155.474
C05221=1061.386,95.175,-75.688,172.038,29.566,155.473
C05222=1061.379,94.926,-75.669,172.036,29.563,155.473
C05223=1061.373,94.642,-75.647,172.035,29.561,155.473
C05224=1061.365,94.357,-75.626,172.033,29.558,155.472
C05225=1061.359,94.072,-75.605,172.031,29.555,155.472
C05226=1061.352,93.788,-75.584,172.030,29.552,155.471
C05227=1061.347,93.539,-75.565,172.028,29.549,155.471
C05228=1061.340,93.289,-75.546,172.026,29.546,155.471
C05229=1061.335,93.040,-75.527,172.025,29.544,155.470
C05230=1061.329,92.792,-75.509,172.023,29.541,155.470
C05231=1061.323,92.542,-75.490,172.022,29.538,155.469
C05232=1061.317,92.292,-75.471,172.020,29.536,155.469
C05233=1061.311,92.043,-75.453,172.019,29.533,155.468
C05234=1061.305,91.795,-75.434,172.017,29.530,155.468
C05235=1061.299,91.545,-75.415,172.015,29.527,155.468
C05236=1061.294,91.295,-75.397,172.015,29.525,155.467
C05237=1061.287,91.046,-75.378,172.013,29.522,155.467
C05238=1061.282,90.798,-75.359,172.011,29.519,155.466
C05239=1061.276,90.548,-75.341,172.010,29.517,155.466
C05240=1061.270,90.299,-75.323,172.008,29.515,155.466
C05241=1061.263,90.050,-75.304,172.006,29.512,155.465
C05242=1061.257,89.800,-75.285,172.005,29.509,155.465
C05243=1061.252,89.551,-75.267,172.004,29.507,155.465
C05244=1061.246,89.302,-75.249,172.002,29.504,155.464
C05245=1061.239,89.053,-75.230,172.000,29.502,155.464
C05246=1061.233,88.803,-75.212,171.999,29.499,155.463
C05247=1061.227,88.554,-75.193,171.998,29.496,155.463
C05248=1061.222,88.305,-75.175,171.996,29.494,155.463
C05249=1061.215,88.056,-75.157,171.995,29.491,155.462
C05250=1061.209,87.806,-75.138,171.993,29.488,155.462
C05251=1061.203,87.557,-75.120,171.991,29.485,155.461
C05252=1061.198,87.308,-75.101,171.989,29.483,155.461
C05253=1061.191,87.059,-75.082,171.989,29.481,155.461
C05254=1061.185,86.809,-75.064,171.987,29.478,155.460
C05255=1061.179,86.561,-75.046,171.985,29.475,155.460
C05256=1061.173,86.311,-75.028,171.984,29.473,155.459
C05257=1061.168,86.061,-75.009,171.982,29.470,155.459
C05258=1061.161,85.812,-74.991,171.981,29.468,155.459
C05259=1061.156,85.563,-74.973,171.980,29.465,155.458
C05260=1061.149,85.314,-74.955,171.978,29.462,155.458
C05261=1061.143,85.064,-74.936,171.976,29.460,155.458
C05262=1061.138,84.816,-74.917,171.975,29.457,155.457
C05263=1061.132,84.566,-74.899,171.973,29.454,155.457
C05264=1061.125,84.317,-74.881,171.972,29.452,155.456
C05265=1061.119,84.067,-74.863,171.970,29.449,155.456
C05266=1061.113,83.819,-74.845,171.969,29.447,155.456
C05267=1061.107,83.569,-74.827,171.967,29.444,155.455
C05268=1061.102,83.319,-74.808,171.965,29.441,155.455
C05269=1061.096,83.070,-74.790,171.965,29.439,155.454
C05270=1061.090,82.821,-74.772,171.963,29.436,155.454
C05271=1061.084,82.572,-74.753,171.961,29.433,155.454
C05272=1061.078,82.323,-74.736,171.960,29.431,155.453
C05273=1061.072,82.073,-74.717,171.958,29.428,155.453
C05274=1061.066,81.824,-74.699,171.957,29.426,155.452
C05275=1061.060,81.575,-74.680,171.956,29.423,155.452
C05276=1061.054,81.325,-74.662,171.954,29.420,155.452
C05277=1061.049,81.076,-74.645,171.952,29.418,155.451
C05278=1061.042,80.827,-74.626,171.950,29.415,155.451
C05279=1061.036,80.577,-74.608,171.950,29.412,155.450
C05280=1061.030,80.329,-74.590,171.948,29.410,155.450
C05281=1061.024,80.079,-74.572,171.946,29.407,155.450
C05282=1061.019,79.830,-74.554,171.945,29.404,155.449
C05283=1061.013,79.581,-74.535,171.943,29.401,155.449
C05284=1061.007,79.331,-74.517,171.942,29.399,155.449
C05285=1061.001,79.082,-74.500,171.941,29.397,155.448
C05286=1060.995,78.833,-74.481,171.939,29.394,155.448
C05287=1060.988,78.548,-74.461,171.937,29.391,155.447
C05288=1060.982,78.264,-74.440,171.936,29.388,155.447
C05289=1060.975,77.980,-74.419,171.934,29.385,155.446
C05290=1060.968,77.695,-74.399,171.932,29.382,155.446
C05291=1060.963,77.446,-74.381,171.931,29.379,155.446
C05292=1060.956,77.197,-74.363,171.929,29.377,155.445
C05293=1060.950,76.947,-74.345,171.927,29.374,155.445
C05294=1060.944,76.698,-74.327,171.927,29.372,155.444
C05295=1060.938,76.449,-74.310,171.925,29.369,155.444
C05296=1060.932,76.200,-74.292,171.923,29.366,155.444
C05297=1060.926,75.951,-74.274,171.922,29.363,155.443
C05298=1060.920,75.701,-74.256,171.920,29.361,155.443
C05299=1060.914,75.452,-74.238,171.919,29.359,155.442
C05300=1060.908,75.202,-74.220,171.917,29.356,155.442
C05301=1060.902,74.954,-74.202,171.916,29.353,155.442
C05302=1060.896,74.704,-74.184,171.914,29.350,155.441
C05303=1060.890,74.455,-74.167,171.912,29.348,155.441
C05304=1060.884,74.205,-74.149,171.912,29.346,155.441
C05305=1060.877,73.956,-74.131,171.910,29.343,155.440
C05306=1060.872,73.707,-74.114,171.908,29.340,155.440
C05307=1060.865,73.457,-74.095,171.907,29.337,155.439
C05308=1060.860,73.208,-74.077,171.905,29.335,155.439
C05309=1060.854,72.959,-74.060,171.904,29.333,155.439
C05310=1060.848,72.710,-74.042,171.903,29.330,155.438
C05311=1060.842,72.460,-74.024,171.901,29.327,155.438
C05312=1060.836,72.211,-74.007,171.899,29.324,155.437
C05313=1060.830,71.961,-73.989,171.898,29.322,155.437
C05314=1060.824,71.712,-73.972,171.897,29.319,155.437
C05315=1060.818,71.463,-73.954,171.895,29.317,155.436
C05316=1060.812,71.214,-73.935,171.893,29.314,155.436
C05317=1060.806,70.965,-73.917,171.892,29.311,155.436
C05318=1060.800,70.716,-73.900,171.890,29.309,155.435
C05319=1060.794,70.466,-73.883,171.889,29.306,155.435
C05320=1060.788,70.217,-73.865,171.888,29.303,155.434
C05321=1060.782,69.967,-73.847,171.886,29.301,155.434
C05322=1060.777,69.718,-73.829,171.884,29.299,155.434
C05323=1060.770,69.469,-73.812,171.883,29.296,155.433
C05324=1060.764,69.220,-73.795,171.882,29.293,155.433
C05325=1060.758,68.970,-73.777,171.880,29.290,155.432
C05326=1060.753,68.721,-73.759,171.879,29.288,155.432
C05327=1060.746,68.472,-73.742,171.877,29.286,155.432
C05328=1060.740,68.223,-73.724,171.875,29.283,155.431
C05329=1060.734,67.973,-73.706,171.875,29.280,155.431
C05330=1060.728,67.724,-73.689,171.873,29.278,155.431
C05331=1060.722,67.474,-73.671,171.871,29.275,155.430
C05332=1060.717,67.225,-73.654,171.870,29.273,155.430
C05333=1060.710,66.975,-73.637,171.868,29.270,155.429
C05334=1060.704,66.726,-73.620,171.867,29.267,155.429
C05335=1060.698,66.476,-73.602,171.865,29.265,155.429
C05336=1060.692,66.228,-73.585,171.864,29.262,155.428
C05337=1060.686,65.978,-73.567,171.862,29.260,155.428
C05338=1060.680,65.729,-73.549,171.861,29.257,155.428
C05339=1060.674,65.480,-73.532,171.860,29.254,155.427
C05340=1060.668,65.230,-73.514,171.858,29.252,155.427
C05341=1060.662,64.981,-73.497,171.856,29.249,155.426
C05342=1060.656,64.731,-73.480,171.855,29.247,155.426
C05343=1060.650,64.482,-73.462,171.854,29.244,155.426
C05344=1060.644,64.233,-73.445,171.852,29.242,155.425
C05345=1060.638,63.984,-73.428,171.851,29.239,155.425
C05346=1060.631,63.734,-73.410,171.849,29.236,155.425
C05347=1060.626,63.485,-73.393,171.847,29.234,155.424
C05348=1060.619,63.235,-73.376,171.847,29.232,155.424
C05349=1060.613,62.986,-73.358,171.845,29.229,155.423
C05350=1060.607,62.737,-73.341,171.843,29.227,155.423
C05351=1060.600,62.453,-73.322,171.842,29.223,155.423
C05352=1060.593,62.168,-73.302,171.840,29.221,155.422
C05353=1060.586,61.884,-73.283,171.838,29.218,155.422
C05354=1060.579,61.600,-73.263,171.837,29.215,155.421
C05355=1060.573,61.349,-73.246,171.835,29.212,155.421
C05356=1060.567,61.100,-73.229,171.833,29.210,155.421
C05357=1060.561,60.851,-73.211,171.832,29.207,155.420
C05358=1060.554,60.601,-73.194,171.831,29.205,155.420
C05359=1060.548,60.353,-73.177,171.829,29.202,155.420
C05360=1060.542,60.103,-73.160,171.828,29.200,155.419
C05361=1060.536,59.853,-73.143,171.826,29.197,155.419
C05362=1060.529,59.604,-73.126,171.824,29.194,155.418
C05363=1060.524,59.355,-73.108,171.823,29.192,155.418
C05364=1060.517,59.106,-73.091,171.822,29.190,155.418
C05365=1060.512,58.856,-73.074,171.820,29.187,155.417
C05366=1060.505,58.607,-73.057,171.818,29.185,155.417
C05367=1060.499,58.358,-73.041,171.817,29.182,155.417
C05368=1060.493,58.108,-73.023,171.816,29.179,155.416
C05369=1060.487,57.859,-73.006,171.814,29.177,155.416
C05370=1060.481,57.609,-72.989,171.813,29.174,155.416
C05371=1060.475,57.360,-72.972,171.811,29.172,155.415
C05372=1060.469,57.111,-72.956,171.809,29.169,155.415
C05373=1060.463,56.861,-72.938,171.809,29.167,155.414
C05374=1060.457,56.612,-72.921,171.807,29.164,155.414
C05375=1060.451,56.363,-72.904,171.805,29.161,155.414
C05376=1060.445,56.113,-72.887,171.804,29.159,155.413
C05377=1060.439,55.864,-72.870,171.802,29.156,155.413
C05378=1060.432,55.615,-72.853,171.801,29.154,155.413
C05379=1060.427,55.365,-72.836,171.800,29.152,155.412
C05380=1060.420,55.116,-72.819,171.798,29.149,155.412
C05381=1060.414,54.868,-72.802,171.796,29.146,155.412
C05382=1060.408,54.617,-72.785,171.795,29.143,155.411
C05383=1060.402,54.368,-72.768,171.794,29.141,155.411
C05384=1060.396,54.119,-72.752,171.792,29.139,155.410
C05385=1060.390,53.869,-72.734,171.791,29.136,155.410
C05386=1060.384,53.620,-72.717,171.789,29.134,155.410
C05387=1060.378,53.371,-72.701,171.788,29.131,155.409
C05388=1060.373,53.122,-72.684,171.787,29.128,155.409
C05389=1060.366,52.872,-72.667,171.785,29.126,155.409
C05390=1060.360,52.623,-72.650,171.783,29.124,155.408
C05391=1060.354,52.373,-72.633,171.782,29.121,155.408
C05392=1060.348,52.124,-72.616,171.781,29.118,155.407
C05393=1060.342,51.874,-72.600,171.779,29.115,155.407
C05394=1060.336,51.625,-72.582,171.777,29.113,155.407
C05395=1060.330,51.376,-72.566,171.776,29.110,155.406
C05396=1060.323,51.127,-72.548,171.774,29.108,155.406
C05397=1060.318,50.877,-72.532,171.773,29.105,155.406
C05398=1060.312,50.628,-72.515,171.772,29.103,155.405
C05399=1060.306,50.379,-72.498,171.770,29.100,155.405
C05400=1060.300,50.129,-72.482,171.768,29.097,155.404
C05401=1060.294,49.879,-72.465,171.767,29.095,155.404
C05402=1060.288,49.630,-72.448,171.766,29.093,155.404
C05403=1060.282,49.381,-72.432,171.764,29.090,155.403
C05404=1060.276,49.132,-72.414,171.763,29.087,155.403
C05405=1060.270,48.882,-72.397,171.761,29.085,155.403
C05406=1060.264,48.633,-72.381,171.760,29.082,155.402
C05407=1060.258,48.384,-72.364,171.759,29.080,155.402
C05408=1060.252,48.134,-72.347,171.757,29.077,155.401
C05409=1060.247,47.885,-72.331,171.755,29.075,155.401
C05410=1060.241,47.636,-72.315,171.754,29.072,155.401
C05411=1060.234,47.386,-72.297,171.753,29.069,155.400
C05412=1060.228,47.136,-72.281,171.751,29.067,155.400
C05413=1060.223,46.887,-72.264,171.750,29.064,155.400
C05414=1060.216,46.638,-72.247,171.748,29.062,155.399
C05415=1060.210,46.353,-72.228,171.746,29.059,155.399
C05416=1060.203,46.068,-72.209,171.745,29.055,155.398
C05417=1060.196,45.784,-72.190,171.743,29.053,155.398
C05418=1060.189,45.499,-72.171,171.742,29.050,155.398
C05419=1060.183,45.250,-72.155,171.740,29.047,155.397
C05420=1060.178,45.000,-72.138,171.739,29.045,155.397
C05421=1060.172,44.751,-72.122,171.738,29.042,155.396
C05422=1060.166,44.501,-72.106,171.736,29.040,155.396
C05423=1060.159,44.252,-72.088,171.734,29.037,155.396
C05424=1060.154,44.002,-72.071,171.733,29.034,155.395
C05425=1060.148,43.753,-72.055,171.732,29.032,155.395
C05426=1060.142,43.504,-72.039,171.730,29.029,155.395
C05427=1060.136,43.254,-72.023,171.729,29.027,155.394
C05428=1060.130,43.005,-72.006,171.727,29.024,155.394
C05429=1060.124,42.756,-71.989,171.725,29.022,155.394
C05430=1060.117,42.506,-71.973,171.725,29.019,155.393
C05431=1060.112,42.257,-71.957,171.723,29.016,155.393
C05432=1060.106,42.007,-71.940,171.721,29.014,155.392
C05433=1060.100,41.758,-71.924,171.720,29.011,155.392
C05434=1060.094,41.509,-71.908,171.718,29.009,155.392
C05435=1060.088,41.259,-71.892,171.717,29.007,155.391
C05436=1060.082,41.010,-71.875,171.716,29.004,155.391
C05437=1060.075,40.760,-71.859,171.714,29.002,155.391
C05438=1060.069,40.511,-71.842,171.712,28.999,155.390
C05439=1060.063,40.262,-71.825,171.711,28.996,155.390
C05440=1060.057,40.013,-71.809,171.710,28.994,155.390
C05441=1060.051,39.763,-71.793,171.708,28.991,155.389
C05442=1060.045,39.514,-71.777,171.707,28.988,155.389
C05443=1060.039,39.265,-71.760,171.705,28.986,155.388
